KUKA KRL program: EPS_2_251349_MH88A_A_20250929014700.src

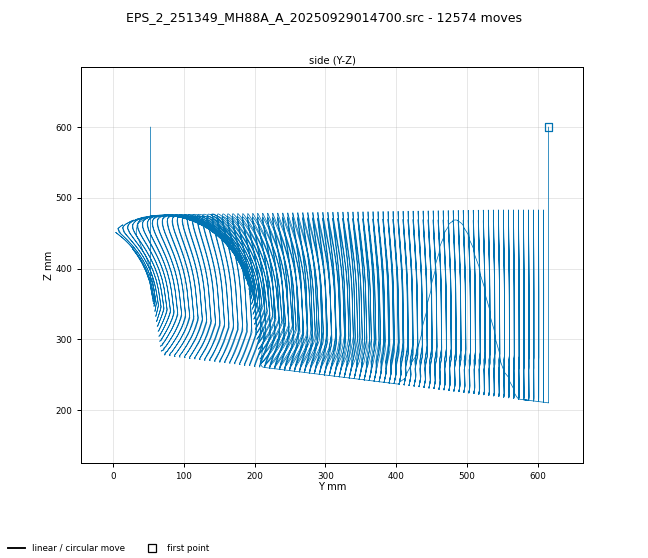
[picture p0: tool path of EPS_2_251349_MH88A_A_20250929014700.src, 12574 of 12576 moves have a stored position in this frame; points joined in program order, loops and branches not executed]
&ACCESS RVP
&REL 4
&COMMENT QRS 19112012
&PARAM EDITMASK = *
DEF PART()
EXT BAS (BAS_COMMAND :IN,REAL :IN )
INT I
BAS (#INITMOV,0 )

;KUKA QRS Post kuka4.cps  Date:22-06-2017 !

File_ID=2863

QRS_PRE_INIT()

;Init var - Until changes are made in qrs_pre_init
Outlet_Square_prg=0
Inlet_1_Square_prg=0
Inlet_2_Square_prg=0
Inlet_3_Square_prg=0
Inlet_4_Square_prg=0
Inlet_5_Square_prg=0

Outlet_1={X 0.000, Y 540.910, Z 382.500, B 0.000, E1 0.000 }
Inlet_1={X 0.000, Y 541.980, Z 367.500, B 0.000, E1 136.000 }
Outlet_1_type=201
Inlet_1_type=201
;QRS#1=Sidecore dimensions
;QRS#2=200-8" PVC SDR 35
;QRS#3=200-8" PVC SDR 35
;QRS#4=
;QRS#5=
;QRS#6=
;QRS#7=
;QRS#8=
;QRS#9=12-08 PSX
;QRS#10=12-08 PSX
;QRS#11=
;QRS#12=
;QRS#13=
;QRS#14=
;QRS#15=
;QRS#16=1220x127x762 2,5'
;QRS#17=EPS Height
;QRS#18=483
;QRS#19=*
;QRS#20= UPDATED VERSION 22-06-2017
;QRS#21=*
Outlet_Square=0100
Inlet_1_Square=0100
Inlet_2_Square=0
Inlet_3_Square=0
Inlet_4_Square=0
Inlet_5_Square=0
Mill_Square=1
Outlet_Square_Prg=204
Inlet_1_Square_prg=204

QRS_INIT()

$ADVANCE=5

; T1
PTP {E1 173.638,E2 173.638}
PTP {X 0,Y 615.435,A -85,B 0,C 180,E1 173.638,E2 173.638,E3 0,E4 0,E5 0,E6 0}
QRS_SPEED_INIT()
LIN {X 0,Y 615.435,Z 600,A -85,B 0,C 180,E1 173.638,E2 173.638,E3 0,E4 0,E5 0,E6 0} C_VEL
LIN {X 0,Y 615.435,Z 220.373,A -85,B 0,C 180,E1 173.638,E2 173.638} C_VEL
LIN {X 0,Y 615.435,Z 212.194,A -85,B 0,C 180,E1 173.638,E2 173.638} C_VEL
LIN {X 0,Y 615.43,Z 210.194,A -85,B 0,C 180,E1 173.452,E2 173.452} C_VEL
LIN {X 0,Y 615.434,Z 210.193,A -85,B 0,C 180,E1 171.468,E2 171.468} C_VEL
LIN {X 0,Y 615.439,Z 210.195,A -85,B 0,C 180,E1 169.126,E2 169.126} C_VEL
LIN {X 0,Y 615.455,Z 210.197,A -85,B 0,C 180,E1 166.803,E2 166.803} C_VEL
LIN {X 0,Y 615.495,Z 210.192,A -85,B 0,C 180,E1 164.101,E2 164.101} C_VEL
LIN {X 0,Y 615.456,Z 210.188,A -85,B 0,C 180,E1 161.359,E2 161.359} C_VEL
LIN {X 0,Y 615.456,Z 210.188,A -85,B 0,C 180,E1 159.274,E2 159.274} C_VEL
LIN {X 0,Y 615.456,Z 210.188,A -85,B 0,C 180,E1 157.161,E2 157.161} C_VEL
LIN {X 0,Y 615.455,Z 210.188,A -85,B 0,C 180,E1 155.013,E2 155.013} C_VEL
LIN {X 0,Y 615.492,Z 210.435,A -85,B 0,C 180,E1 154.019,E2 154.019} C_VEL
LIN {X 0,Y 615.489,Z 227.308,A -85,B 0,C 180,E1 151.349,E2 151.349} C_VEL
LIN {X 0,Y 615.432,Z 244.946,A -85,B 0,C 180,E1 148.617,E2 148.617} C_VEL
LIN {X 0,Y 615.462,Z 256.479,A -85,B 0,C 180,E1 146.868,E2 146.868} C_VEL
LIN {X 0,Y 615.457,Z 258.435,A -85,B 0,C 180,E1 146.794,E2 146.794} C_VEL
LIN {X 0,Y 615.498,Z 364.416,A -85,B 0,C 180,E1 145.533,E2 145.533} C_VEL
LIN {X 0,Y 615.498,Z 377.381,A -85,B 0,C 180,E1 145.244,E2 145.244} C_VEL
LIN {X 0,Y 615.498,Z 389.548,A -85,B 0,C 180,E1 144.844,E2 144.844} C_VEL
LIN {X 0,Y 615.482,Z 401.088,A -85,B 0,C 180,E1 144.335,E2 144.335} C_VEL
LIN {X 0,Y 615.475,Z 412.93,A -85,B 0,C 180,E1 143.656,E2 143.656} C_VEL
LIN {X 0,Y 615.498,Z 423.238,A -85,B 0,C 180,E1 142.913,E2 142.913} C_VEL
LIN {X 0,Y 615.495,Z 431.49,A -85,B 0,C 180,E1 142.181,E2 142.181} C_VEL
LIN {X 0,Y 615.496,Z 439.782,A -85,B 0,C 180,E1 141.315,E2 141.315} C_VEL
LIN {X 0,Y 615.497,Z 447.794,A -85,B 0,C 180,E1 140.26,E2 140.26} C_VEL
LIN {X 0,Y 615.496,Z 454.438,A -85,B 0,C 180,E1 139.154,E2 139.154} C_VEL
LIN {X 0,Y 615.495,Z 458.784,A -85,B 0,C 180,E1 138.227,E2 138.227} C_VEL
LIN {X 0,Y 615.494,Z 462.154,A -85,B 0,C 180,E1 137.304,E2 137.304} C_VEL
LIN {X 0,Y 615.493,Z 465.473,A -85,B 0,C 180,E1 136,E2 136} C_VEL
LIN {X 0,Y 615.493,Z 466.94,A -85,B 0,C 180,E1 134.942,E2 134.942} C_VEL
LIN {X 0,Y 615.492,Z 467.383,A -85,B 0,C 180,E1 134.008,E2 134.008} C_VEL
LIN {X 0,Y 615.489,Z 467.004,A -85,B 0,C 180,E1 133.058,E2 133.058} C_VEL
LIN {X 0,Y 615.494,Z 465.774,A -85,B 0,C 180,E1 132.092,E2 132.092} C_VEL
LIN {X 0,Y 615.495,Z 463.616,A -85,B 0,C 180,E1 131.106,E2 131.106} C_VEL
LIN {X 0,Y 615.497,Z 460.421,A -85,B 0,C 180,E1 130.101,E2 130.101} C_VEL
LIN {X 0,Y 615.493,Z 455.189,A -85,B 0,C 180,E1 128.902,E2 128.902} C_VEL
LIN {X 0,Y 615.494,Z 448.993,A -85,B 0,C 180,E1 127.828,E2 127.828} C_VEL
LIN {X 0,Y 615.495,Z 441.609,A -85,B 0,C 180,E1 126.818,E2 126.818} C_VEL
LIN {X 0,Y 615.497,Z 434.167,A -85,B 0,C 180,E1 125.991,E2 125.991} C_VEL
LIN {X 0,Y 615.498,Z 424.68,A -85,B 0,C 180,E1 125.112,E2 125.112} C_VEL
LIN {X 0,Y 615.494,Z 414.65,A -85,B 0,C 180,E1 124.367,E2 124.367} C_VEL
LIN {X 0,Y 615.48,Z 402.826,A -85,B 0,C 180,E1 123.666,E2 123.666} C_VEL
LIN {X 0,Y 615.497,Z 391.367,A -85,B 0,C 180,E1 123.136,E2 123.136} C_VEL
LIN {X 0,Y 615.498,Z 378.544,A -85,B 0,C 180,E1 122.698,E2 122.698} C_VEL
LIN {X 0,Y 615.497,Z 365.74,A -85,B 0,C 180,E1 122.401,E2 122.401} C_VEL
LIN {X 0,Y 615.477,Z 340.468,A -85,B 0,C 180,E1 122.078,E2 122.078} C_VEL
LIN {X 0,Y 615.431,Z 257.305,A -85,B 0,C 180,E1 121.092,E2 121.092} C_VEL
LIN {X 0,Y 615.435,Z 256.163,A -85,B 0,C 180,E1 121.006,E2 121.006} C_VEL
LIN {X 0,Y 615.491,Z 239.577,A -85,B 0,C 180,E1 118.467,E2 118.467} C_VEL
LIN {X 0,Y 615.479,Z 221.082,A -85,B 0,C 180,E1 115.585,E2 115.585} C_VEL
LIN {X 0,Y 615.488,Z 210.314,A -85,B 0,C 180,E1 113.851,E2 113.851} C_VEL
LIN {X 0,Y 615.454,Z 210.199,A -85,B 0,C 180,E1 111.432,E2 111.432} C_VEL
LIN {X 0,Y 615.451,Z 210.199,A -85,B 0,C 180,E1 109.338,E2 109.338} C_VEL
LIN {X 0,Y 615.448,Z 210.2,A -85,B 0,C 180,E1 107.27,E2 107.27} C_VEL
LIN {X 0,Y 615.408,Z 210.198,A -85,B 0,C 180,E1 104.55,E2 104.55} C_VEL
LIN {X 0,Y 615.407,Z 210.199,A -85,B 0,C 180,E1 102.53,E2 102.53} C_VEL
LIN {X 0,Y 615.408,Z 210.199,A -85,B 0,C 180,E1 100.527,E2 100.527} C_VEL
LIN {X 0,Y 615.41,Z 210.199,A -85,B 0,C 180,E1 98.536,E2 98.536} C_VEL
LIN {X 0,Y 615.414,Z 210.199,A -85,B 0,C 180,E1 96.556,E2 96.556} C_VEL
LIN {X 0,Y 615.421,Z 210.2,A -85,B 0,C 180,E1 94.584,E2 94.584} C_VEL
LIN {X 0,Y 615.43,Z 210.2,A -85,B 0,C 180,E1 92.617,E2 92.617} C_VEL
LIN {X 0,Y 615.441,Z 210.2,A -85,B 0,C 180,E1 90.653,E2 90.653} C_VEL
LIN {X 0,Y 615.402,Z 210.2,A -85,B 0,C 180,E1 88.036,E2 88.036} C_VEL
LIN {X 0,Y 615.406,Z 210.2,A -85,B 0,C 180,E1 86.07,E2 86.07} C_VEL
LIN {X 0,Y 615.412,Z 210.199,A -85,B 0,C 180,E1 84.1,E2 84.1} C_VEL
LIN {X 0,Y 615.42,Z 210.199,A -85,B 0,C 180,E1 82.123,E2 82.123} C_VEL
LIN {X 0,Y 615.429,Z 210.199,A -85,B 0,C 180,E1 80.136,E2 80.136} C_VEL
LIN {X 0,Y 615.438,Z 210.198,A -85,B 0,C 180,E1 78.137,E2 78.137} C_VEL
LIN {X 0,Y 615.438,Z 210.198,A -85,B 0,C 180,E1 76.052,E2 76.052} C_VEL
LIN {X 0,Y 615.407,Z 210.199,A -85,B 0,C 180,E1 73.41,E2 73.41} C_VEL
LIN {X 0,Y 615.408,Z 210.198,A -85,B 0,C 180,E1 71.351,E2 71.351} C_VEL
LIN {X 0,Y 615.407,Z 210.199,A -85,B 0,C 180,E1 69.266,E2 69.266} C_VEL
LIN {X 0,Y 615.408,Z 210.198,A -85,B 0,C 180,E1 67.151,E2 67.151} C_VEL
LIN {X 0,Y 615.412,Z 210.198,A -85,B 0,C 180,E1 65.004,E2 65.004} C_VEL
LIN {X 0,Y 615.48,Z 210.203,A -85,B 0,C 180,E1 62.084,E2 62.084} C_VEL
LIN {X 0,Y 615.499,Z 210.195,A -85,B 0,C 180,E1 59.84,E2 59.84} C_VEL
LIN {X 0,Y 615.468,Z 210.194,A -85,B 0,C 180,E1 57.541,E2 57.541} C_VEL
LIN {X 0,Y 615.436,Z 210.195,A -85,B 0,C 180,E1 55.181,E2 55.181} C_VEL
LIN {X 0,Y 615.418,Z 210.196,A -85,B 0,C 180,E1 52.752,E2 52.752} C_VEL
LIN {X 0,Y 615.457,Z 210.199,A -85,B 0,C 180,E1 49.903,E2 49.903} C_VEL
LIN {X 0,Y 615.446,Z 210.194,A -85,B 0,C 180,E1 46.946,E2 46.946} C_VEL
LIN {X 0,Y 615.424,Z 210.197,A -85,B 0,C 180,E1 44.145,E2 44.145} C_VEL
LIN {X 0,Y 615.425,Z 210.196,A -85,B 0,C 180,E1 42.073,E2 42.073} C_VEL
LIN {X 0,Y 615.44,Z 210.198,A -85,B 0,C 180,E1 39.745,E2 39.745} C_VEL
LIN {X 0,Y 615.487,Z 210.193,A -85,B 0,C 180,E1 36.936,E2 36.936} C_VEL
LIN {X 0,Y 615.477,Z 210.191,A -85,B 0,C 180,E1 34.698,E2 34.698} C_VEL
LIN {X 0,Y 615.444,Z 210.192,A -85,B 0,C 180,E1 32.324,E2 32.324} C_VEL
LIN {X 0,Y 615.438,Z 210.192,A -85,B 0,C 180,E1 30.155,E2 30.155} C_VEL
LIN {X 0,Y 615.431,Z 210.193,A -85,B 0,C 180,E1 27.911,E2 27.911} C_VEL
LIN {X 0,Y 615.429,Z 210.195,A -85,B 0,C 180,E1 25.557,E2 25.557} C_VEL
LIN {X 0,Y 615.481,Z 210.199,A -85,B 0,C 180,E1 22.838,E2 22.838} C_VEL
LIN {X 0,Y 615.465,Z 210.189,A -85,B 0,C 180,E1 20.028,E2 20.028} C_VEL
LIN {X 0,Y 615.461,Z 210.19,A -85,B 0,C 180,E1 17.952,E2 17.952} C_VEL
LIN {X 0,Y 615.469,Z 210.189,A -85,B 0,C 180,E1 15.9,E2 15.9} C_VEL
LIN {X 0,Y 615.475,Z 210.188,A -85,B 0,C 180,E1 13.869,E2 13.869} C_VEL
LIN {X 0,Y 615.433,Z 210.193,A -85,B 0,C 180,E1 11.189,E2 11.189} C_VEL
LIN {X 0,Y 615.437,Z 210.192,A -85,B 0,C 180,E1 9.195,E2 9.195} C_VEL
LIN {X 0,Y 615.441,Z 210.191,A -85,B 0,C 180,E1 7.211,E2 7.211} C_VEL
LIN {X 0,Y 615.447,Z 210.19,A -85,B 0,C 180,E1 5.237,E2 5.237} C_VEL
LIN {X 0,Y 615.456,Z 210.188,A -85,B 0,C 180,E1 3.269,E2 3.269} C_VEL
LIN {X 0,Y 615.468,Z 210.187,A -85,B 0,C 180,E1 1.304,E2 1.304} C_VEL
LIN {X 0,Y 615.439,Z 210.192,A -85,B 0,C 180,E1 -1.313,E2 -1.313} C_VEL
LIN {X 0,Y 615.466,Z 210.197,A -85,B 0,C 180,E1 -3.933,E2 -3.933} C_VEL
LIN {X 0,Y 615.493,Z 210.19,A -85,B 0,C 180,E1 -6.58,E2 -6.58} C_VEL
LIN {X 0,Y 615.46,Z 210.187,A -85,B 0,C 180,E1 -9.203,E2 -9.203} C_VEL
LIN {X 0,Y 615.468,Z 210.186,A -85,B 0,C 180,E1 -11.197,E2 -11.197} C_VEL
LIN {X 0,Y 615.474,Z 210.186,A -85,B 0,C 180,E1 -13.205,E2 -13.205} C_VEL
LIN {X 0,Y 615.482,Z 210.184,A -85,B 0,C 180,E1 -15.23,E2 -15.23} C_VEL
LIN {X 0,Y 615.446,Z 210.192,A -85,B 0,C 180,E1 -17.961,E2 -17.961} C_VEL
LIN {X 0,Y 615.489,Z 210.201,A -85,B 0,C 180,E1 -20.734,E2 -20.734} C_VEL
LIN {X 0,Y 615.48,Z 210.184,A -85,B 0,C 180,E1 -23.56,E2 -23.56} C_VEL
LIN {X 0,Y 615.474,Z 210.184,A -85,B 0,C 180,E1 -25.719,E2 -25.719} C_VEL
LIN {X 0,Y 615.464,Z 210.186,A -85,B 0,C 180,E1 -27.919,E2 -27.919} C_VEL
LIN {X 0,Y 615.455,Z 210.188,A -85,B 0,C 180,E1 -30.165,E2 -30.165} C_VEL
LIN {X 0,Y 615.451,Z 210.191,A -85,B 0,C 180,E1 -32.462,E2 -32.462} C_VEL
LIN {X 0,Y 615.459,Z 210.194,A -85,B 0,C 180,E1 -34.819,E2 -34.819} C_VEL
LIN {X 0,Y 615.484,Z 210.2,A -85,B 0,C 180,E1 -37.245,E2 -37.245} C_VEL
LIN {X 0,Y 615.496,Z 210.181,A -85,B 0,C 180,E1 -40.089,E2 -40.089} C_VEL
LIN {X 0,Y 615.473,Z 210.184,A -85,B 0,C 180,E1 -42.356,E2 -42.356} C_VEL
LIN {X 0,Y 615.455,Z 210.193,A -85,B 0,C 180,E1 -45.074,E2 -45.074} C_VEL
LIN {X 0,Y 615.487,Z 210.194,A -85,B 0,C 180,E1 -47.922,E2 -47.922} C_VEL
LIN {X 0,Y 615.49,Z 210.186,A -85,B 0,C 180,E1 -50.249,E2 -50.249} C_VEL
LIN {X 0,Y 615.478,Z 210.183,A -85,B 0,C 180,E1 -52.756,E2 -52.756} C_VEL
LIN {X 0,Y 615.458,Z 210.19,A -85,B 0,C 180,E1 -55.305,E2 -55.305} C_VEL
LIN {X 0,Y 615.466,Z 210.195,A -85,B 0,C 180,E1 -57.674,E2 -57.674} C_VEL
LIN {X 0,Y 615.494,Z 210.197,A -85,B 0,C 180,E1 -60.206,E2 -60.206} C_VEL
LIN {X 0,Y 615.497,Z 210.179,A -85,B 0,C 180,E1 -62.955,E2 -62.955} C_VEL
LIN {X 0,Y 615.462,Z 210.19,A -85,B 0,C 180,E1 -65.726,E2 -65.726} C_VEL
LIN {X 0,Y 615.489,Z 210.311,A -85,B 0,C 180,E1 -68.435,E2 -68.435} C_VEL
LIN {X 0,Y 615.496,Z 213.29,A -85,B 0,C 180,E1 -68.919,E2 -68.919} C_VEL
LIN {X 0,Y 615.486,Z 233.846,A -85,B 0,C 180,E1 -71.881,E2 -71.881} C_VEL
LIN {X 0,Y 615.474,Z 253.027,A -85,B 0,C 180,E1 -74.603,E2 -74.603} C_VEL
LIN {X 0,Y 615.487,Z 270.928,A -85,B 0,C 180,E1 -77.092,E2 -77.092} C_VEL
LIN {X 0,Y 615.488,Z 272.814,A -85,B 0,C 180,E1 -77.155,E2 -77.155} C_VEL
LIN {X 0,Y 615.498,Z 378.773,A -85,B 0,C 180,E1 -78.41,E2 -78.41} C_VEL
LIN {X 0,Y 615.498,Z 391.306,A -85,B 0,C 180,E1 -78.681,E2 -78.681} C_VEL
LIN {X 0,Y 615.496,Z 404.523,A -85,B 0,C 180,E1 -79.11,E2 -79.11} C_VEL
LIN {X 0,Y 615.491,Z 416.457,A -85,B 0,C 180,E1 -79.638,E2 -79.638} C_VEL
LIN {X 0,Y 615.48,Z 427.981,A -85,B 0,C 180,E1 -80.303,E2 -80.303} C_VEL
LIN {X 0,Y 615.499,Z 438.328,A -85,B 0,C 180,E1 -81.049,E2 -81.049} C_VEL
LIN {X 0,Y 615.497,Z 446.681,A -85,B 0,C 180,E1 -81.793,E2 -81.793} C_VEL
LIN {X 0,Y 615.498,Z 454.597,A -85,B 0,C 180,E1 -82.619,E2 -82.619} C_VEL
LIN {X 0,Y 615.49,Z 462.197,A -85,B 0,C 180,E1 -83.607,E2 -83.607} C_VEL
LIN {X 0,Y 615.498,Z 469.199,A -85,B 0,C 180,E1 -84.758,E2 -84.758} C_VEL
LIN {X 0,Y 615.493,Z 473.847,A -85,B 0,C 180,E1 -85.743,E2 -85.743} C_VEL
LIN {X 0,Y 615.494,Z 477.395,A -85,B 0,C 180,E1 -86.726,E2 -86.726} C_VEL
LIN {X 0,Y 615.497,Z 479.23,A -85,B 0,C 180,E1 -87.381,E2 -87.381} C_VEL
LIN {X 0,Y 615.497,Z 480.606,A -85,B 0,C 180,E1 -88.036,E2 -88.036} C_VEL
LIN {X 0,Y 615.496,Z 482.173,A -85,B 0,C 180,E1 -89.345,E2 -89.345} C_VEL
LIN {X 0,Y 615.494,Z 482.389,A -85,B 0,C 180,E1 -89.999,E2 -89.999} C_VEL
LIN {X 0,Y 615.495,Z 481.581,A -85,B 0,C 180,E1 -91.307,E2 -91.307} C_VEL
LIN {X 0,Y 615.497,Z 480.61,A -85,B 0,C 180,E1 -91.962,E2 -91.962} C_VEL
LIN {X 0,Y 615.497,Z 479.236,A -85,B 0,C 180,E1 -92.617,E2 -92.617} C_VEL
LIN {X 0,Y 615.496,Z 476.353,A -85,B 0,C 180,E1 -93.599,E2 -93.599} C_VEL
LIN {X 0,Y 615.498,Z 472.446,A -85,B 0,C 180,E1 -94.583,E2 -94.583} C_VEL
LIN {X 0,Y 615.499,Z 467.411,A -85,B 0,C 180,E1 -95.568,E2 -95.568} C_VEL
LIN {X 0,Y 615.489,Z 460.921,A -85,B 0,C 180,E1 -96.577,E2 -96.577} C_VEL
LIN {X 0,Y 615.497,Z 453.144,A -85,B 0,C 180,E1 -97.544,E2 -97.544} C_VEL
LIN {X 0,Y 615.498,Z 443.272,A -85,B 0,C 180,E1 -98.535,E2 -98.535} C_VEL
LIN {X 0,Y 615.495,Z 432.883,A -85,B 0,C 180,E1 -99.363,E2 -99.363} C_VEL
LIN {X 0,Y 615.475,Z 422.599,A -85,B 0,C 180,E1 -100.027,E2 -100.027} C_VEL
LIN {X 0,Y 615.497,Z 411.121,A -85,B 0,C 180,E1 -100.617,E2 -100.617} C_VEL
LIN {X 0,Y 615.499,Z 399.3,A -85,B 0,C 180,E1 -101.079,E2 -101.079} C_VEL
LIN {X 0,Y 615.498,Z 386.295,A -85,B 0,C 180,E1 -101.442,E2 -101.442} C_VEL
LIN {X 0,Y 615.5,Z 373.041,A -85,B 0,C 180,E1 -101.671,E2 -101.671} C_VEL
LIN {X 0,Y 615.488,Z 271.781,A -85,B 0,C 180,E1 -102.864,E2 -102.864} C_VEL
LIN {X 0,Y 615.485,Z 270.529,A -85,B 0,C 180,E1 -102.948,E2 -102.948} C_VEL
LIN {X 0,Y 615.481,Z 250.637,A -85,B 0,C 180,E1 -105.734,E2 -105.734} C_VEL
LIN {X 0,Y 615.491,Z 231.59,A -85,B 0,C 180,E1 -108.442,E2 -108.442} C_VEL
LIN {X 0,Y 615.492,Z 212.102,A -85,B 0,C 180,E1 -111.255,E2 -111.255} C_VEL
LIN {X 0,Y 615.49,Z 210.317,A -85,B 0,C 180,E1 -111.562,E2 -111.562} C_VEL
LIN {X 0,Y 615.461,Z 210.191,A -85,B 0,C 180,E1 -114.272,E2 -114.272} C_VEL
LIN {X 0,Y 615.457,Z 210.189,A -85,B 0,C 180,E1 -116.444,E2 -116.444} C_VEL
LIN {X 0,Y 615.459,Z 210.188,A -85,B 0,C 180,E1 -118.658,E2 -118.658} C_VEL
LIN {X 0,Y 615.485,Z 210.183,A -85,B 0,C 180,E1 -121.084,E2 -121.084} C_VEL
LIN {X 0,Y 615.483,Z 210.2,A -85,B 0,C 180,E1 -124.02,E2 -124.02} C_VEL
LIN {X 0,Y 615.456,Z 210.195,A -85,B 0,C 180,E1 -126.425,E2 -126.425} C_VEL
LIN {X 0,Y 615.453,Z 210.188,A -85,B 0,C 180,E1 -129.056,E2 -129.056} C_VEL
LIN {X 0,Y 615.479,Z 210.186,A -85,B 0,C 180,E1 -131.472,E2 -131.472} C_VEL
LIN {X 0,Y 615.495,Z 210.201,A -85,B 0,C 180,E1 -134.147,E2 -134.147} C_VEL
LIN {X 0,Y 615.443,Z 210.196,A -85,B 0,C 180,E1 -136.749,E2 -136.749} C_VEL
LIN {X 0,Y 615.438,Z 210.195,A -85,B 0,C 180,E1 -138.908,E2 -138.908} C_VEL
LIN {X 0,Y 615.432,Z 210.195,A -85,B 0,C 180,E1 -141.089,E2 -141.089} C_VEL
LIN {X 0,Y 615.439,Z 210.193,A -85,B 0,C 180,E1 -143.57,E2 -143.57} C_VEL
LIN {X 0,Y 615.467,Z 210.192,A -85,B 0,C 180,E1 -145.974,E2 -145.974} C_VEL
LIN {X 0,Y 615.445,Z 210.198,A -85,B 0,C 180,E1 -148.917,E2 -148.917} C_VEL
LIN {X 0,Y 615.418,Z 210.198,A -85,B 0,C 180,E1 -151.336,E2 -151.336} C_VEL
LIN {X 0,Y 615.414,Z 210.197,A -85,B 0,C 180,E1 -153.55,E2 -153.55} C_VEL
LIN {X 0,Y 615.425,Z 210.197,A -85,B 0,C 180,E1 -156,E2 -156} C_VEL
LIN {X 0,Y 615.48,Z 210.197,A -85,B 0,C 180,E1 -158.565,E2 -158.565} C_VEL
LIN {X 0,Y 615.419,Z 210.2,A -85,B 0,C 180,E1 -161.408,E2 -161.408} C_VEL
LIN {X 0,Y 615.41,Z 210.2,A -85,B 0,C 180,E1 -163.587,E2 -163.587} C_VEL
LIN {X 0,Y 615.424,Z 210.2,A -85,B 0,C 180,E1 -165.446,E2 -165.446} C_VEL
LIN {X 0,Y 615.433,Z 210.199,A -85,B 0,C 180,E1 -167.465,E2 -167.465} C_VEL
LIN {X 0,Y 615.442,Z 210.198,A -85,B 0,C 180,E1 -169.469,E2 -169.469} C_VEL
LIN {X 0,Y 615.412,Z 210.198,A -85,B 0,C 180,E1 -172.12,E2 -172.12} C_VEL
LIN {X 0,Y 615.416,Z 210.197,A -85,B 0,C 180,E1 -174.097,E2 -174.097} C_VEL
LIN {X 0,Y 615.421,Z 210.196,A -85,B 0,C 180,E1 -176.067,E2 -176.067} C_VEL
LIN {X 0,Y 615.429,Z 210.195,A -85,B 0,C 180,E1 -178.033,E2 -178.033} C_VEL
LIN {X 0,Y 615.438,Z 210.194,A -85,B 0,C 180,E1 -179.996,E2 -179.996} C_VEL
LIN {X 0,Y 615.449,Z 210.192,A -85,B 0,C 180,E1 -181.959,E2 -181.959} C_VEL
LIN {X 0,Y 615.462,Z 210.191,A -85,B 0,C 180,E1 -183.924,E2 -183.924} C_VEL
LIN {X 0,Y 615.43,Z 210.194,A -85,B 0,C 180,E1 -186.548,E2 -186.548} C_VEL
LIN {X 0,Y 614.774,Z 210.348,A -85,B 0,C 180,E1 -187.094,E2 -187.094} C_VEL
LIN {X 0,Y 611.95,Z 210.753,A -85,B 0,C 180,E1 -187.98,E2 -187.98} C_VEL
LIN {X 0,Y 609.559,Z 211.067,A -85,B 0,C 180,E1 -188.693,E2 -188.693} C_VEL
LIN {X 0,Y 608.529,Z 211.186,A -85,B 0,C 180,E1 -189.243,E2 -189.243} C_VEL
LIN {X 0,Y 608.444,Z 211.194,A -85,B 0,C 180,E1 -189.429,E2 -189.429} C_VEL
LIN {X 0,Y 608.456,Z 211.19,A -85,B 0,C 180,E1 -191.995,E2 -191.995} C_VEL
LIN {X 0,Y 608.44,Z 211.188,A -85,B 0,C 180,E1 -194.716,E2 -194.716} C_VEL
LIN {X 0,Y 608.442,Z 211.188,A -85,B 0,C 180,E1 -196.779,E2 -196.779} C_VEL
LIN {X 0,Y 608.434,Z 211.197,A -85,B 0,C 180,E1 -199.565,E2 -199.565} C_VEL
LIN {X 0,Y 608.46,Z 211.187,A -85,B 0,C 180,E1 -202.481,E2 -202.481} C_VEL
LIN {X 0,Y 608.438,Z 211.19,A -85,B 0,C 180,E1 -204.565,E2 -204.565} C_VEL
LIN {X 0,Y 608.493,Z 211.364,A -85,B 0,C 180,E1 -205.884,E2 -205.884} C_VEL
LIN {X 0,Y 608.508,Z 227.357,A -85,B 0,C 180,E1 -208.441,E2 -208.441} C_VEL
LIN {X 0,Y 608.429,Z 245.716,A -85,B 0,C 180,E1 -211.311,E2 -211.311} C_VEL
LIN {X 0,Y 608.473,Z 256.851,A -85,B 0,C 180,E1 -213.006,E2 -213.006} C_VEL
LIN {X 0,Y 608.548,Z 258.93,A -85,B 0,C 180,E1 -213.063,E2 -213.063} C_VEL
LIN {X 0,Y 608.571,Z 364.391,A -85,B 0,C 180,E1 -214.33,E2 -214.33} C_VEL
LIN {X 0,Y 608.552,Z 378.116,A -85,B 0,C 180,E1 -214.642,E2 -214.642} C_VEL
LIN {X 0,Y 608.525,Z 390.367,A -85,B 0,C 180,E1 -215.056,E2 -215.056} C_VEL
LIN {X 0,Y 608.488,Z 401.771,A -85,B 0,C 180,E1 -215.571,E2 -215.571} C_VEL
LIN {X 0,Y 608.484,Z 412.397,A -85,B 0,C 180,E1 -216.184,E2 -216.184} C_VEL
LIN {X 0,Y 608.472,Z 422.516,A -85,B 0,C 180,E1 -216.905,E2 -216.905} C_VEL
LIN {X 0,Y 608.476,Z 430.315,A -85,B 0,C 180,E1 -217.578,E2 -217.578} C_VEL
LIN {X 0,Y 608.452,Z 438.224,A -85,B 0,C 180,E1 -218.383,E2 -218.383} C_VEL
LIN {X 0,Y 608.437,Z 446.625,A -85,B 0,C 180,E1 -219.433,E2 -219.433} C_VEL
LIN {X 0,Y 608.433,Z 453.423,A -85,B 0,C 180,E1 -220.513,E2 -220.513} C_VEL
LIN {X 0,Y 608.446,Z 459.075,A -85,B 0,C 180,E1 -221.67,E2 -221.67} C_VEL
LIN {X 0,Y 608.457,Z 461.663,A -85,B 0,C 180,E1 -222.336,E2 -222.336} C_VEL
LIN {X 0,Y 608.428,Z 464.571,A -85,B 0,C 180,E1 -223.307,E2 -223.307} C_VEL
LIN {X 0,Y 608.418,Z 466.54,A -85,B 0,C 180,E1 -224.263,E2 -224.263} C_VEL
LIN {X 0,Y 608.414,Z 467.657,A -85,B 0,C 180,E1 -225.203,E2 -225.203} C_VEL
LIN {X 0,Y 608.419,Z 467.987,A -85,B 0,C 180,E1 -226.128,E2 -226.128} C_VEL
LIN {X 0,Y 608.424,Z 467.549,A -85,B 0,C 180,E1 -227.04,E2 -227.04} C_VEL
LIN {X 0,Y 608.421,Z 466.357,A -85,B 0,C 180,E1 -227.938,E2 -227.938} C_VEL
LIN {X 0,Y 608.429,Z 464.462,A -85,B 0,C 180,E1 -228.823,E2 -228.823} C_VEL
LIN {X 0,Y 608.442,Z 461.86,A -85,B 0,C 180,E1 -229.698,E2 -229.698} C_VEL
LIN {X 0,Y 608.435,Z 457.896,A -85,B 0,C 180,E1 -230.695,E2 -230.695} C_VEL
LIN {X 0,Y 608.434,Z 452.449,A -85,B 0,C 180,E1 -231.752,E2 -231.752} C_VEL
LIN {X 0,Y 608.437,Z 445.317,A -85,B 0,C 180,E1 -232.833,E2 -232.833} C_VEL
LIN {X 0,Y 608.469,Z 438.226,A -85,B 0,C 180,E1 -233.706,E2 -233.706} C_VEL
LIN {X 0,Y 608.478,Z 428.002,A -85,B 0,C 180,E1 -234.727,E2 -234.727} C_VEL
LIN {X 0,Y 608.484,Z 417.879,A -85,B 0,C 180,E1 -235.534,E2 -235.534} C_VEL
LIN {X 0,Y 608.474,Z 406.727,A -85,B 0,C 180,E1 -236.251,E2 -236.251} C_VEL
LIN {X 0,Y 608.518,Z 395.236,A -85,B 0,C 180,E1 -236.83,E2 -236.83} C_VEL
LIN {X 0,Y 608.533,Z 382.108,A -85,B 0,C 180,E1 -237.328,E2 -237.328} C_VEL
LIN {X 0,Y 608.562,Z 369.579,A -85,B 0,C 180,E1 -237.661,E2 -237.661} C_VEL
LIN {X 0,Y 608.57,Z 356.478,A -85,B 0,C 180,E1 -237.872,E2 -237.872} C_VEL
LIN {X 0,Y 608.462,Z 257.306,A -85,B 0,C 180,E1 -239.058,E2 -239.058} C_VEL
LIN {X 0,Y 608.442,Z 256.088,A -85,B 0,C 180,E1 -239.175,E2 -239.175} C_VEL
LIN {X 0,Y 608.486,Z 237.153,A -85,B 0,C 180,E1 -242.112,E2 -242.112} C_VEL
LIN {X 0,Y 608.503,Z 219.537,A -85,B 0,C 180,E1 -244.886,E2 -244.886} C_VEL
LIN {X 0,Y 608.481,Z 211.305,A -85,B 0,C 180,E1 -246.225,E2 -246.225} C_VEL
LIN {X 0,Y 608.392,Z 211.195,A -85,B 0,C 180,E1 -249.018,E2 -249.018} C_VEL
LIN {X 0,Y 608.404,Z 211.195,A -85,B 0,C 180,E1 -251.828,E2 -251.828} C_VEL
LIN {X 0,Y 608.434,Z 211.198,A -85,B 0,C 180,E1 -254.595,E2 -254.595} C_VEL
LIN {X 0,Y 608.407,Z 211.193,A -85,B 0,C 180,E1 -257.323,E2 -257.323} C_VEL
LIN {X 0,Y 608.394,Z 211.195,A -85,B 0,C 180,E1 -259.35,E2 -259.35} C_VEL
LIN {X 0,Y 608.389,Z 211.196,A -85,B 0,C 180,E1 -261.364,E2 -261.364} C_VEL
LIN {X 0,Y 608.391,Z 211.196,A -85,B 0,C 180,E1 -263.368,E2 -263.368} C_VEL
LIN {X 0,Y 608.394,Z 211.196,A -85,B 0,C 180,E1 -265.363,E2 -265.363} C_VEL
LIN {X 0,Y 608.421,Z 211.194,A -85,B 0,C 180,E1 -267.353,E2 -267.353} C_VEL
LIN {X 0,Y 608.389,Z 211.194,A -85,B 0,C 180,E1 -270.001,E2 -270.001} C_VEL
LIN {X 0,Y 608.419,Z 211.194,A -85,B 0,C 180,E1 -272.649,E2 -272.649} C_VEL
LIN {X 0,Y 608.47,Z 211.194,A -85,B 0,C 180,E1 -275.303,E2 -275.303} C_VEL
LIN {X 0,Y 608.408,Z 211.193,A -85,B 0,C 180,E1 -277.969,E2 -277.969} C_VEL
LIN {X 0,Y 608.394,Z 211.195,A -85,B 0,C 180,E1 -279.979,E2 -279.979} C_VEL
LIN {X 0,Y 608.403,Z 211.194,A -85,B 0,C 180,E1 -282.002,E2 -282.002} C_VEL
LIN {X 0,Y 608.405,Z 211.193,A -85,B 0,C 180,E1 -284.723,E2 -284.723} C_VEL
LIN {X 0,Y 608.413,Z 211.201,A -85,B 0,C 180,E1 -287.479,E2 -287.479} C_VEL
LIN {X 0,Y 608.41,Z 211.194,A -85,B 0,C 180,E1 -290.277,E2 -290.277} C_VEL
LIN {X 0,Y 608.39,Z 211.195,A -85,B 0,C 180,E1 -292.481,E2 -292.481} C_VEL
LIN {X 0,Y 608.397,Z 211.194,A -85,B 0,C 180,E1 -294.574,E2 -294.574} C_VEL
LIN {X 0,Y 608.409,Z 211.193,A -85,B 0,C 180,E1 -297.212,E2 -297.212} C_VEL
LIN {X 0,Y 608.473,Z 211.195,A -85,B 0,C 180,E1 -299.988,E2 -299.988} C_VEL
LIN {X 0,Y 608.407,Z 211.193,A -85,B 0,C 180,E1 -302.883,E2 -302.883} C_VEL
LIN {X 0,Y 608.387,Z 211.194,A -85,B 0,C 180,E1 -305.282,E2 -305.282} C_VEL
LIN {X 0,Y 608.437,Z 211.199,A -85,B 0,C 180,E1 -308.249,E2 -308.249} C_VEL
LIN {X 0,Y 608.459,Z 211.197,A -85,B 0,C 180,E1 -310.341,E2 -310.341} C_VEL
LIN {X 0,Y 608.418,Z 211.194,A -85,B 0,C 180,E1 -312.964,E2 -312.964} C_VEL
LIN {X 0,Y 608.398,Z 211.193,A -85,B 0,C 180,E1 -315.743,E2 -315.743} C_VEL
LIN {X 0,Y 608.405,Z 211.193,A -85,B 0,C 180,E1 -317.943,E2 -317.943} C_VEL
LIN {X 0,Y 608.458,Z 211.197,A -85,B 0,C 180,E1 -320.705,E2 -320.705} C_VEL
LIN {X 0,Y 608.454,Z 211.192,A -85,B 0,C 180,E1 -323.093,E2 -323.093} C_VEL
LIN {X 0,Y 608.443,Z 211.189,A -85,B 0,C 180,E1 -325.537,E2 -325.537} C_VEL
LIN {X 0,Y 608.421,Z 211.19,A -85,B 0,C 180,E1 -327.911,E2 -327.911} C_VEL
LIN {X 0,Y 608.413,Z 211.191,A -85,B 0,C 180,E1 -330.225,E2 -330.225} C_VEL
LIN {X 0,Y 608.433,Z 211.194,A -85,B 0,C 180,E1 -332.802,E2 -332.802} C_VEL
LIN {X 0,Y 608.449,Z 211.188,A -85,B 0,C 180,E1 -335.855,E2 -335.855} C_VEL
LIN {X 0,Y 608.429,Z 211.189,A -85,B 0,C 180,E1 -338.313,E2 -338.313} C_VEL
LIN {X 0,Y 608.411,Z 211.191,A -85,B 0,C 180,E1 -340.434,E2 -340.434} C_VEL
LIN {X 0,Y 608.41,Z 211.191,A -85,B 0,C 180,E1 -342.528,E2 -342.528} C_VEL
LIN {X 0,Y 608.431,Z 211.189,A -85,B 0,C 180,E1 -344.599,E2 -344.599} C_VEL
LIN {X 0,Y 608.454,Z 211.192,A -85,B 0,C 180,E1 -347.328,E2 -347.328} C_VEL
LIN {X 0,Y 608.458,Z 211.191,A -85,B 0,C 180,E1 -350.028,E2 -350.028} C_VEL
LIN {X 0,Y 608.42,Z 211.19,A -85,B 0,C 180,E1 -352.705,E2 -352.705} C_VEL
LIN {X 0,Y 608.433,Z 211.189,A -85,B 0,C 180,E1 -354.703,E2 -354.703} C_VEL
LIN {X 0,Y 608.438,Z 211.19,A -85,B 0,C 180,E1 -357.356,E2 -357.356} C_VEL
LIN {X 0,Y 608.474,Z 211.194,A -85,B 0,C 180,E1 -360.004,E2 -360.004} C_VEL
LIN {X 0,Y 608.48,Z 211.186,A -85,B 0,C 180,E1 -362.652,E2 -362.652} C_VEL
LIN {X 0,Y 608.429,Z 211.189,A -85,B 0,C 180,E1 -365.306,E2 -365.306} C_VEL
LIN {X 0,Y 608.426,Z 211.189,A -85,B 0,C 180,E1 -367.304,E2 -367.304} C_VEL
LIN {X 0,Y 608.429,Z 211.193,A -85,B 0,C 180,E1 -369.981,E2 -369.981} C_VEL
LIN {X 0,Y 608.476,Z 211.191,A -85,B 0,C 180,E1 -372.68,E2 -372.68} C_VEL
LIN {X 0,Y 608.458,Z 211.186,A -85,B 0,C 180,E1 -375.41,E2 -375.41} C_VEL
LIN {X 0,Y 608.422,Z 211.193,A -85,B 0,C 180,E1 -378.176,E2 -378.176} C_VEL
LIN {X 0,Y 608.461,Z 211.193,A -85,B 0,C 180,E1 -380.984,E2 -380.984} C_VEL
LIN {X 0,Y 608.442,Z 211.187,A -85,B 0,C 180,E1 -383.849,E2 -383.849} C_VEL
LIN {X 0,Y 608.428,Z 211.189,A -85,B 0,C 180,E1 -386.039,E2 -386.039} C_VEL
LIN {X 0,Y 608.421,Z 211.191,A -85,B 0,C 180,E1 -388.271,E2 -388.271} C_VEL
LIN {X 0,Y 608.435,Z 211.191,A -85,B 0,C 180,E1 -390.549,E2 -390.549} C_VEL
LIN {X 0,Y 608.447,Z 211.193,A -85,B 0,C 180,E1 -392.883,E2 -392.883} C_VEL
LIN {X 0,Y 608.438,Z 211.2,A -85,B 0,C 180,E1 -395.28,E2 -395.28} C_VEL
LIN {X 0,Y 608.469,Z 211.189,A -85,B 0,C 180,E1 -397.749,E2 -397.749} C_VEL
LIN {X 0,Y 608.449,Z 211.187,A -85,B 0,C 180,E1 -400.328,E2 -400.328} C_VEL
LIN {X 0,Y 608.426,Z 211.192,A -85,B 0,C 180,E1 -402.964,E2 -402.964} C_VEL
LIN {X 0,Y 608.457,Z 211.195,A -85,B 0,C 180,E1 -405.738,E2 -405.738} C_VEL
LIN {X 0,Y 608.45,Z 211.187,A -85,B 0,C 180,E1 -408.661,E2 -408.661} C_VEL
LIN {X 0,Y 608.427,Z 211.194,A -85,B 0,C 180,E1 -411.408,E2 -411.408} C_VEL
LIN {X 0,Y 608.453,Z 211.197,A -85,B 0,C 180,E1 -413.956,E2 -413.956} C_VEL
LIN {X 0,Y 608.456,Z 211.191,A -85,B 0,C 180,E1 -416.328,E2 -416.328} C_VEL
LIN {X 0,Y 608.456,Z 211.187,A -85,B 0,C 180,E1 -418.733,E2 -418.733} C_VEL
LIN {X 0,Y 608.455,Z 211.187,A -85,B 0,C 180,E1 -421.385,E2 -421.385} C_VEL
LIN {X 0,Y 608.44,Z 211.194,A -85,B 0,C 180,E1 -423.963,E2 -423.963} C_VEL
LIN {X 0,Y 608.451,Z 211.19,A -85,B 0,C 180,E1 -426.875,E2 -426.875} C_VEL
LIN {X 0,Y 608.471,Z 211.348,A -85,B 0,C 180,E1 -428.352,E2 -428.352} C_VEL
LIN {X 0,Y 608.512,Z 222.951,A -85,B 0,C 180,E1 -430.079,E2 -430.079} C_VEL
LIN {X 0,Y 608.52,Z 242.257,A -85,B 0,C 180,E1 -432.871,E2 -432.871} C_VEL
LIN {X 0,Y 608.482,Z 262.769,A -85,B 0,C 180,E1 -435.791,E2 -435.791} C_VEL
LIN {X 0,Y 608.497,Z 271.281,A -85,B 0,C 180,E1 -436.962,E2 -436.962} C_VEL
LIN {X 0,Y 608.588,Z 276.426,A -85,B 0,C 180,E1 -437.049,E2 -437.049} C_VEL
LIN {X 0,Y 608.549,Z 378.893,A -85,B 0,C 180,E1 -438.276,E2 -438.276} C_VEL
LIN {X 0,Y 608.549,Z 392.181,A -85,B 0,C 180,E1 -438.571,E2 -438.571} C_VEL
LIN {X 0,Y 608.546,Z 405.34,A -85,B 0,C 180,E1 -439.009,E2 -439.009} C_VEL
LIN {X 0,Y 608.516,Z 416.616,A -85,B 0,C 180,E1 -439.518,E2 -439.518} C_VEL
LIN {X 0,Y 608.468,Z 428.182,A -85,B 0,C 180,E1 -440.19,E2 -440.19} C_VEL
LIN {X 0,Y 608.485,Z 438.581,A -85,B 0,C 180,E1 -440.945,E2 -440.945} C_VEL
LIN {X 0,Y 608.459,Z 446.992,A -85,B 0,C 180,E1 -441.698,E2 -441.698} C_VEL
LIN {X 0,Y 608.471,Z 454.951,A -85,B 0,C 180,E1 -442.533,E2 -442.533} C_VEL
LIN {X 0,Y 608.438,Z 462.3,A -85,B 0,C 180,E1 -443.486,E2 -443.486} C_VEL
LIN {X 0,Y 608.45,Z 467.86,A -85,B 0,C 180,E1 -444.365,E2 -444.365} C_VEL
LIN {X 0,Y 608.432,Z 472.945,A -85,B 0,C 180,E1 -445.361,E2 -445.361} C_VEL
LIN {X 0,Y 608.449,Z 476.893,A -85,B 0,C 180,E1 -446.357,E2 -446.357} C_VEL
LIN {X 0,Y 608.425,Z 479.806,A -85,B 0,C 180,E1 -447.351,E2 -447.351} C_VEL
LIN {X 0,Y 608.442,Z 481.199,A -85,B 0,C 180,E1 -448.013,E2 -448.013} C_VEL
LIN {X 0,Y 608.439,Z 482.783,A -85,B 0,C 180,E1 -449.337,E2 -449.337} C_VEL
LIN {X 0,Y 608.434,Z 483,A -85,B 0,C 180,E1 -449.999,E2 -449.999} C_VEL
LIN {X 0,Y 608.448,Z 482.185,A -85,B 0,C 180,E1 -451.323,E2 -451.323} C_VEL
LIN {X 0,Y 608.442,Z 481.203,A -85,B 0,C 180,E1 -451.985,E2 -451.985} C_VEL
LIN {X 0,Y 608.425,Z 479.812,A -85,B 0,C 180,E1 -452.647,E2 -452.647} C_VEL
LIN {X 0,Y 608.449,Z 476.9,A -85,B 0,C 180,E1 -453.641,E2 -453.641} C_VEL
LIN {X 0,Y 608.432,Z 472.955,A -85,B 0,C 180,E1 -454.637,E2 -454.637} C_VEL
LIN {X 0,Y 608.437,Z 466.884,A -85,B 0,C 180,E1 -455.8,E2 -455.8} C_VEL
LIN {X 0,Y 608.461,Z 460.244,A -85,B 0,C 180,E1 -456.798,E2 -456.798} C_VEL
LIN {X 0,Y 608.456,Z 452,A -85,B 0,C 180,E1 -457.799,E2 -457.799} C_VEL
LIN {X 0,Y 608.477,Z 441.613,A -85,B 0,C 180,E1 -458.802,E2 -458.802} C_VEL
LIN {X 0,Y 608.486,Z 430.766,A -85,B 0,C 180,E1 -459.64,E2 -459.64} C_VEL
LIN {X 0,Y 608.489,Z 419.797,A -85,B 0,C 180,E1 -460.312,E2 -460.312} C_VEL
LIN {X 0,Y 608.536,Z 407.809,A -85,B 0,C 180,E1 -460.888,E2 -460.888} C_VEL
LIN {X 0,Y 608.533,Z 395.919,A -85,B 0,C 180,E1 -461.321,E2 -461.321} C_VEL
LIN {X 0,Y 608.542,Z 383.582,A -85,B 0,C 180,E1 -461.638,E2 -461.638} C_VEL
LIN {X 0,Y 608.574,Z 367.844,A -85,B 0,C 180,E1 -461.869,E2 -461.869} C_VEL
LIN {X 0,Y 608.547,Z 271.791,A -85,B 0,C 180,E1 -463.013,E2 -463.013} C_VEL
LIN {X 0,Y 608.459,Z 270.661,A -85,B 0,C 180,E1 -463.1,E2 -463.1} C_VEL
LIN {X 0,Y 608.494,Z 250.72,A -85,B 0,C 180,E1 -465.919,E2 -465.919} C_VEL
LIN {X 0,Y 608.516,Z 231.17,A -85,B 0,C 180,E1 -468.727,E2 -468.727} C_VEL
LIN {X 0,Y 608.549,Z 212.109,A -85,B 0,C 180,E1 -471.509,E2 -471.509} C_VEL
LIN {X 0,Y 608.478,Z 211.266,A -85,B 0,C 180,E1 -471.69,E2 -471.69} C_VEL
LIN {X 0,Y 608.444,Z 211.188,A -85,B 0,C 180,E1 -474.57,E2 -474.57} C_VEL
LIN {X 0,Y 608.486,Z 211.185,A -85,B 0,C 180,E1 -477.207,E2 -477.207} C_VEL
LIN {X 0,Y 608.451,Z 211.195,A -85,B 0,C 180,E1 -479.967,E2 -479.967} C_VEL
LIN {X 0,Y 608.434,Z 211.19,A -85,B 0,C 180,E1 -482.516,E2 -482.516} C_VEL
LIN {X 0,Y 608.423,Z 211.19,A -85,B 0,C 180,E1 -484.9,E2 -484.9} C_VEL
LIN {X 0,Y 608.465,Z 211.192,A -85,B 0,C 180,E1 -487.744,E2 -487.744} C_VEL
LIN {X 0,Y 608.439,Z 211.195,A -85,B 0,C 180,E1 -490.326,E2 -490.326} C_VEL
LIN {X 0,Y 608.413,Z 211.192,A -85,B 0,C 180,E1 -492.961,E2 -492.961} C_VEL
LIN {X 0,Y 608.418,Z 211.191,A -85,B 0,C 180,E1 -495.198,E2 -495.198} C_VEL
LIN {X 0,Y 608.475,Z 211.189,A -85,B 0,C 180,E1 -497.938,E2 -497.938} C_VEL
LIN {X 0,Y 608.419,Z 211.195,A -85,B 0,C 180,E1 -500.706,E2 -500.706} C_VEL
LIN {X 0,Y 608.4,Z 211.194,A -85,B 0,C 180,E1 -503.079,E2 -503.079} C_VEL
LIN {X 0,Y 608.427,Z 211.19,A -85,B 0,C 180,E1 -505.525,E2 -505.525} C_VEL
LIN {X 0,Y 608.435,Z 211.191,A -85,B 0,C 180,E1 -507.901,E2 -507.901} C_VEL
LIN {X 0,Y 608.46,Z 211.191,A -85,B 0,C 180,E1 -510.217,E2 -510.217} C_VEL
LIN {X 0,Y 608.395,Z 211.195,A -85,B 0,C 180,E1 -513.22,E2 -513.22} C_VEL
LIN {X 0,Y 608.404,Z 211.193,A -85,B 0,C 180,E1 -515.424,E2 -515.424} C_VEL
LIN {X 0,Y 608.438,Z 211.192,A -85,B 0,C 180,E1 -518.304,E2 -518.304} C_VEL
LIN {X 0,Y 608.407,Z 211.195,A -85,B 0,C 180,E1 -521.296,E2 -521.296} C_VEL
LIN {X 0,Y 608.386,Z 211.195,A -85,B 0,C 180,E1 -523.901,E2 -523.901} C_VEL
LIN {X 0,Y 608.433,Z 211.195,A -85,B 0,C 180,E1 -526.639,E2 -526.639} C_VEL
LIN {X 0,Y 608.434,Z 211.194,A -85,B 0,C 180,E1 -529.346,E2 -529.346} C_VEL
LIN {X 0,Y 608.385,Z 211.195,A -85,B 0,C 180,E1 -532.028,E2 -532.028} C_VEL
LIN {X 0,Y 608.398,Z 211.193,A -85,B 0,C 180,E1 -534.029,E2 -534.029} C_VEL
LIN {X 0,Y 608.394,Z 211.194,A -85,B 0,C 180,E1 -536.022,E2 -536.022} C_VEL
LIN {X 0,Y 608.403,Z 211.193,A -85,B 0,C 180,E1 -538.01,E2 -538.01} C_VEL
LIN {X 0,Y 608.431,Z 211.19,A -85,B 0,C 180,E1 -539.996,E2 -539.996} C_VEL
LIN {X 0,Y 608.418,Z 211.192,A -85,B 0,C 180,E1 -541.981,E2 -541.981} C_VEL
LIN {X 0,Y 608.428,Z 211.191,A -85,B 0,C 180,E1 -543.97,E2 -543.97} C_VEL
LIN {X 0,Y 608.414,Z 211.192,A -85,B 0,C 180,E1 -546.596,E2 -546.596} C_VEL
LIN {X 0,Y 608.411,Z 211.192,A -85,B 0,C 180,E1 -548.632,E2 -548.632} C_VEL
LIN {X 0,Y 608.444,Z 211.194,A -85,B 0,C 180,E1 -549.429,E2 -549.429} C_VEL
LIN {X 0,Y 607.775,Z 211.274,A -85,B 0,C 180,E1 -549.982,E2 -549.982} C_VEL
LIN {X 0,Y 604.929,Z 211.627,A -85,B 0,C 180,E1 -550.879,E2 -550.879} C_VEL
LIN {X 0,Y 602.521,Z 211.936,A -85,B 0,C 180,E1 -551.6,E2 -551.6} C_VEL
LIN {X 0,Y 601.478,Z 212.058,A -85,B 0,C 180,E1 -552.156,E2 -552.156} C_VEL
LIN {X 0,Y 601.389,Z 212.067,A -85,B 0,C 180,E1 -552.345,E2 -552.345} C_VEL
LIN {X 0,Y 601.398,Z 212.066,A -85,B 0,C 180,E1 -554.892,E2 -554.892} C_VEL
LIN {X 0,Y 601.402,Z 212.066,A -85,B 0,C 180,E1 -556.981,E2 -556.981} C_VEL
LIN {X 0,Y 601.391,Z 212.077,A -85,B 0,C 180,E1 -559.804,E2 -559.804} C_VEL
LIN {X 0,Y 601.42,Z 212.063,A -85,B 0,C 180,E1 -562.676,E2 -562.676} C_VEL
LIN {X 0,Y 601.381,Z 212.07,A -85,B 0,C 180,E1 -564.873,E2 -564.873} C_VEL
LIN {X 0,Y 601.458,Z 212.24,A -85,B 0,C 180,E1 -565.78,E2 -565.78} C_VEL
LIN {X 0,Y 601.482,Z 223.309,A -85,B 0,C 180,E1 -567.581,E2 -567.581} C_VEL
LIN {X 0,Y 601.412,Z 238.271,A -85,B 0,C 180,E1 -569.961,E2 -569.961} C_VEL
LIN {X 0,Y 601.433,Z 256.579,A -85,B 0,C 180,E1 -572.826,E2 -572.826} C_VEL
LIN {X 0,Y 601.625,Z 258.311,A -85,B 0,C 180,E1 -572.903,E2 -572.903} C_VEL
LIN {X 0,Y 601.611,Z 364.783,A -85,B 0,C 180,E1 -574.2,E2 -574.2} C_VEL
LIN {X 0,Y 601.596,Z 377.988,A -85,B 0,C 180,E1 -574.505,E2 -574.505} C_VEL
LIN {X 0,Y 601.557,Z 390.029,A -85,B 0,C 180,E1 -574.914,E2 -574.914} C_VEL
LIN {X 0,Y 601.502,Z 402.483,A -85,B 0,C 180,E1 -575.487,E2 -575.487} C_VEL
LIN {X 0,Y 601.476,Z 412.957,A -85,B 0,C 180,E1 -576.105,E2 -576.105} C_VEL
LIN {X 0,Y 601.452,Z 423.601,A -85,B 0,C 180,E1 -576.884,E2 -576.884} C_VEL
LIN {X 0,Y 601.43,Z 431.769,A -85,B 0,C 180,E1 -577.622,E2 -577.622} C_VEL
LIN {X 0,Y 601.393,Z 439.765,A -85,B 0,C 180,E1 -578.469,E2 -578.469} C_VEL
LIN {X 0,Y 601.378,Z 447.814,A -85,B 0,C 180,E1 -579.531,E2 -579.531} C_VEL
LIN {X 0,Y 601.344,Z 454.073,A -85,B 0,C 180,E1 -580.568,E2 -580.568} C_VEL
LIN {X 0,Y 601.362,Z 459.677,A -85,B 0,C 180,E1 -581.761,E2 -581.761} C_VEL
LIN {X 0,Y 601.353,Z 462.867,A -85,B 0,C 180,E1 -582.666,E2 -582.666} C_VEL
LIN {X 0,Y 601.33,Z 465.295,A -85,B 0,C 180,E1 -583.585,E2 -583.585} C_VEL
LIN {X 0,Y 601.331,Z 466.974,A -85,B 0,C 180,E1 -584.529,E2 -584.529} C_VEL
LIN {X 0,Y 601.332,Z 467.852,A -85,B 0,C 180,E1 -585.476,E2 -585.476} C_VEL
LIN {X 0,Y 601.327,Z 467.918,A -85,B 0,C 180,E1 -586.427,E2 -586.427} C_VEL
LIN {X 0,Y 601.337,Z 467.154,A -85,B 0,C 180,E1 -587.406,E2 -587.406} C_VEL
LIN {X 0,Y 601.344,Z 465.509,A -85,B 0,C 180,E1 -588.404,E2 -588.404} C_VEL
LIN {X 0,Y 601.332,Z 462.866,A -85,B 0,C 180,E1 -589.425,E2 -589.425} C_VEL
LIN {X 0,Y 601.349,Z 459.111,A -85,B 0,C 180,E1 -590.463,E2 -590.463} C_VEL
LIN {X 0,Y 601.339,Z 454.04,A -85,B 0,C 180,E1 -591.528,E2 -591.528} C_VEL
LIN {X 0,Y 601.381,Z 447.458,A -85,B 0,C 180,E1 -592.612,E2 -592.612} C_VEL
LIN {X 0,Y 601.383,Z 439.962,A -85,B 0,C 180,E1 -593.598,E2 -593.598} C_VEL
LIN {X 0,Y 601.423,Z 432.265,A -85,B 0,C 180,E1 -594.419,E2 -594.419} C_VEL
LIN {X 0,Y 601.436,Z 424.008,A -85,B 0,C 180,E1 -595.173,E2 -595.173} C_VEL
LIN {X 0,Y 601.466,Z 412.763,A -85,B 0,C 180,E1 -595.998,E2 -595.998} C_VEL
LIN {X 0,Y 601.496,Z 402.684,A -85,B 0,C 180,E1 -596.593,E2 -596.593} C_VEL
LIN {X 0,Y 601.556,Z 390.27,A -85,B 0,C 180,E1 -597.166,E2 -597.166} C_VEL
LIN {X 0,Y 601.59,Z 377.654,A -85,B 0,C 180,E1 -597.595,E2 -597.595} C_VEL
LIN {X 0,Y 601.618,Z 363.903,A -85,B 0,C 180,E1 -597.906,E2 -597.906} C_VEL
LIN {X 0,Y 601.451,Z 257.415,A -85,B 0,C 180,E1 -599.208,E2 -599.208} C_VEL
LIN {X 0,Y 601.421,Z 256.656,A -85,B 0,C 180,E1 -599.255,E2 -599.255} C_VEL
LIN {X 0,Y 601.483,Z 238.205,A -85,B 0,C 180,E1 -602.138,E2 -602.138} C_VEL
LIN {X 0,Y 601.508,Z 221.748,A -85,B 0,C 180,E1 -604.758,E2 -604.758} C_VEL
LIN {X 0,Y 601.421,Z 212.222,A -85,B 0,C 180,E1 -606.317,E2 -606.317} C_VEL
LIN {X 0,Y 601.36,Z 212.071,A -85,B 0,C 180,E1 -609.197,E2 -609.197} C_VEL
LIN {X 0,Y 601.361,Z 212.071,A -85,B 0,C 180,E1 -611.608,E2 -611.608} C_VEL
LIN {X 0,Y 601.38,Z 212.078,A -85,B 0,C 180,E1 -614.409,E2 -614.409} C_VEL
LIN {X 0,Y 601.36,Z 212.072,A -85,B 0,C 180,E1 -617.172,E2 -617.172} C_VEL
LIN {X 0,Y 601.369,Z 212.069,A -85,B 0,C 180,E1 -619.905,E2 -619.905} C_VEL
LIN {X 0,Y 601.4,Z 212.074,A -85,B 0,C 180,E1 -622.616,E2 -622.616} C_VEL
LIN {X 0,Y 601.366,Z 212.072,A -85,B 0,C 180,E1 -625.309,E2 -625.309} C_VEL
LIN {X 0,Y 601.386,Z 212.071,A -85,B 0,C 180,E1 -627.322,E2 -627.322} C_VEL
LIN {X 0,Y 601.358,Z 212.07,A -85,B 0,C 180,E1 -630.001,E2 -630.001} C_VEL
LIN {X 0,Y 601.384,Z 212.071,A -85,B 0,C 180,E1 -632.68,E2 -632.68} C_VEL
LIN {X 0,Y 601.421,Z 212.07,A -85,B 0,C 180,E1 -635.365,E2 -635.365} C_VEL
LIN {X 0,Y 601.369,Z 212.069,A -85,B 0,C 180,E1 -638.063,E2 -638.063} C_VEL
LIN {X 0,Y 601.358,Z 212.072,A -85,B 0,C 180,E1 -640.778,E2 -640.778} C_VEL
LIN {X 0,Y 601.372,Z 212.079,A -85,B 0,C 180,E1 -643.518,E2 -643.518} C_VEL
LIN {X 0,Y 601.386,Z 212.067,A -85,B 0,C 180,E1 -646.289,E2 -646.289} C_VEL
LIN {X 0,Y 601.355,Z 212.073,A -85,B 0,C 180,E1 -649.102,E2 -649.102} C_VEL
LIN {X 0,Y 601.363,Z 212.077,A -85,B 0,C 180,E1 -651.962,E2 -651.962} C_VEL
LIN {X 0,Y 601.4,Z 212.068,A -85,B 0,C 180,E1 -654.304,E2 -654.304} C_VEL
LIN {X 0,Y 601.383,Z 212.067,A -85,B 0,C 180,E1 -657.115,E2 -657.115} C_VEL
LIN {X 0,Y 601.432,Z 212.07,A -85,B 0,C 180,E1 -660.165,E2 -660.165} C_VEL
LIN {X 0,Y 601.378,Z 212.068,A -85,B 0,C 180,E1 -663.317,E2 -663.317} C_VEL
LIN {X 0,Y 601.395,Z 212.077,A -85,B 0,C 180,E1 -666.273,E2 -666.273} C_VEL
LIN {X 0,Y 601.362,Z 212.07,A -85,B 0,C 180,E1 -669.131,E2 -669.131} C_VEL
LIN {X 0,Y 601.377,Z 212.069,A -85,B 0,C 180,E1 -671.77,E2 -671.77} C_VEL
LIN {X 0,Y 601.375,Z 212.079,A -85,B 0,C 180,E1 -674.541,E2 -674.541} C_VEL
LIN {X 0,Y 601.371,Z 212.069,A -85,B 0,C 180,E1 -677.336,E2 -677.336} C_VEL
LIN {X 0,Y 601.372,Z 212.069,A -85,B 0,C 180,E1 -680.011,E2 -680.011} C_VEL
LIN {X 0,Y 601.407,Z 212.072,A -85,B 0,C 180,E1 -682.622,E2 -682.622} C_VEL
LIN {X 0,Y 601.426,Z 212.069,A -85,B 0,C 180,E1 -685.077,E2 -685.077} C_VEL
LIN {X 0,Y 601.401,Z 212.067,A -85,B 0,C 180,E1 -687.49,E2 -687.49} C_VEL
LIN {X 0,Y 601.375,Z 212.068,A -85,B 0,C 180,E1 -689.861,E2 -689.861} C_VEL
LIN {X 0,Y 601.373,Z 212.068,A -85,B 0,C 180,E1 -692.137,E2 -692.137} C_VEL
LIN {X 0,Y 601.371,Z 212.069,A -85,B 0,C 180,E1 -694.386,E2 -694.386} C_VEL
LIN {X 0,Y 601.368,Z 212.07,A -85,B 0,C 180,E1 -696.594,E2 -696.594} C_VEL
LIN {X 0,Y 601.428,Z 212.07,A -85,B 0,C 180,E1 -699.204,E2 -699.204} C_VEL
LIN {X 0,Y 601.41,Z 212.072,A -85,B 0,C 180,E1 -701.614,E2 -701.614} C_VEL
LIN {X 0,Y 601.383,Z 212.067,A -85,B 0,C 180,E1 -704.414,E2 -704.414} C_VEL
LIN {X 0,Y 601.395,Z 212.069,A -85,B 0,C 180,E1 -707.177,E2 -707.177} C_VEL
LIN {X 0,Y 601.43,Z 212.069,A -85,B 0,C 180,E1 -709.91,E2 -709.91} C_VEL
LIN {X 0,Y 601.393,Z 212.066,A -85,B 0,C 180,E1 -712.619,E2 -712.619} C_VEL
LIN {X 0,Y 601.404,Z 212.065,A -85,B 0,C 180,E1 -714.641,E2 -714.641} C_VEL
LIN {X 0,Y 601.407,Z 212.065,A -85,B 0,C 180,E1 -717.325,E2 -717.325} C_VEL
LIN {X 0,Y 601.443,Z 212.07,A -85,B 0,C 180,E1 -720.004,E2 -720.004} C_VEL
LIN {X 0,Y 601.442,Z 212.062,A -85,B 0,C 180,E1 -722.683,E2 -722.683} C_VEL
LIN {X 0,Y 601.396,Z 212.065,A -85,B 0,C 180,E1 -725.368,E2 -725.368} C_VEL
LIN {X 0,Y 601.378,Z 212.068,A -85,B 0,C 180,E1 -727.39,E2 -727.39} C_VEL
LIN {X 0,Y 601.395,Z 212.071,A -85,B 0,C 180,E1 -730.099,E2 -730.099} C_VEL
LIN {X 0,Y 601.417,Z 212.068,A -85,B 0,C 180,E1 -732.832,E2 -732.832} C_VEL
LIN {X 0,Y 601.397,Z 212.065,A -85,B 0,C 180,E1 -735.595,E2 -735.595} C_VEL
LIN {X 0,Y 601.383,Z 212.067,A -85,B 0,C 180,E1 -737.692,E2 -737.692} C_VEL
LIN {X 0,Y 601.392,Z 212.066,A -85,B 0,C 180,E1 -739.813,E2 -739.813} C_VEL
LIN {X 0,Y 601.418,Z 212.07,A -85,B 0,C 180,E1 -742.605,E2 -742.605} C_VEL
LIN {X 0,Y 601.418,Z 212.064,A -85,B 0,C 180,E1 -745.621,E2 -745.621} C_VEL
LIN {X 0,Y 601.377,Z 212.068,A -85,B 0,C 180,E1 -747.872,E2 -747.872} C_VEL
LIN {X 0,Y 601.413,Z 212.063,A -85,B 0,C 180,E1 -750.168,E2 -750.168} C_VEL
LIN {X 0,Y 601.406,Z 212.068,A -85,B 0,C 180,E1 -752.712,E2 -752.712} C_VEL
LIN {X 0,Y 601.386,Z 212.075,A -85,B 0,C 180,E1 -755.11,E2 -755.11} C_VEL
LIN {X 0,Y 601.444,Z 212.069,A -85,B 0,C 180,E1 -757.421,E2 -757.421} C_VEL
LIN {X 0,Y 601.414,Z 212.063,A -85,B 0,C 180,E1 -760.572,E2 -760.572} C_VEL
LIN {X 0,Y 601.382,Z 212.067,A -85,B 0,C 180,E1 -762.675,E2 -762.675} C_VEL
LIN {X 0,Y 601.414,Z 212.072,A -85,B 0,C 180,E1 -765.48,E2 -765.48} C_VEL
LIN {X 0,Y 601.423,Z 212.063,A -85,B 0,C 180,E1 -768.409,E2 -768.409} C_VEL
LIN {X 0,Y 601.399,Z 212.065,A -85,B 0,C 180,E1 -770.872,E2 -770.872} C_VEL
LIN {X 0,Y 601.394,Z 212.069,A -85,B 0,C 180,E1 -773.416,E2 -773.416} C_VEL
LIN {X 0,Y 601.426,Z 212.071,A -85,B 0,C 180,E1 -776.067,E2 -776.067} C_VEL
LIN {X 0,Y 601.428,Z 212.064,A -85,B 0,C 180,E1 -778.546,E2 -778.546} C_VEL
LIN {X 0,Y 601.414,Z 212.064,A -85,B 0,C 180,E1 -781.371,E2 -781.371} C_VEL
LIN {X 0,Y 601.4,Z 212.067,A -85,B 0,C 180,E1 -783.635,E2 -783.635} C_VEL
LIN {X 0,Y 601.422,Z 212.067,A -85,B 0,C 180,E1 -785.857,E2 -785.857} C_VEL
LIN {X 0,Y 601.453,Z 212.238,A -85,B 0,C 180,E1 -788.222,E2 -788.222} C_VEL
LIN {X 0,Y 601.612,Z 218.342,A -85,B 0,C 180,E1 -789.158,E2 -789.158} C_VEL
LIN {X 0,Y 601.53,Z 237.431,A -85,B 0,C 180,E1 -791.963,E2 -791.963} C_VEL
LIN {X 0,Y 601.451,Z 255.53,A -85,B 0,C 180,E1 -794.582,E2 -794.582} C_VEL
LIN {X 0,Y 601.461,Z 271.279,A -85,B 0,C 180,E1 -796.807,E2 -796.807} C_VEL
LIN {X 0,Y 601.67,Z 274.637,A -85,B 0,C 180,E1 -796.876,E2 -796.876} C_VEL
LIN {X 0,Y 601.621,Z 378.893,A -85,B 0,C 180,E1 -798.139,E2 -798.139} C_VEL
LIN {X 0,Y 601.593,Z 392.182,A -85,B 0,C 180,E1 -798.437,E2 -798.437} C_VEL
LIN {X 0,Y 601.552,Z 403.918,A -85,B 0,C 180,E1 -798.826,E2 -798.826} C_VEL
LIN {X 0,Y 601.531,Z 414.903,A -85,B 0,C 180,E1 -799.31,E2 -799.31} C_VEL
LIN {X 0,Y 601.462,Z 425.564,A -85,B 0,C 180,E1 -799.904,E2 -799.904} C_VEL
LIN {X 0,Y 601.447,Z 436.463,A -85,B 0,C 180,E1 -800.668,E2 -800.668} C_VEL
LIN {X 0,Y 601.424,Z 445.308,A -85,B 0,C 180,E1 -801.43,E2 -801.43} C_VEL
LIN {X 0,Y 601.397,Z 453.468,A -85,B 0,C 180,E1 -802.276,E2 -802.276} C_VEL
LIN {X 0,Y 601.384,Z 461.463,A -85,B 0,C 180,E1 -803.288,E2 -803.288} C_VEL
LIN {X 0,Y 601.372,Z 467.86,A -85,B 0,C 180,E1 -804.298,E2 -804.298} C_VEL
LIN {X 0,Y 601.336,Z 472.945,A -85,B 0,C 180,E1 -805.306,E2 -805.306} C_VEL
LIN {X 0,Y 601.368,Z 476.892,A -85,B 0,C 180,E1 -806.314,E2 -806.314} C_VEL
LIN {X 0,Y 601.325,Z 479.806,A -85,B 0,C 180,E1 -807.319,E2 -807.319} C_VEL
LIN {X 0,Y 601.341,Z 481.2,A -85,B 0,C 180,E1 -807.99,E2 -807.99} C_VEL
LIN {X 0,Y 601.339,Z 482.783,A -85,B 0,C 180,E1 -809.329,E2 -809.329} C_VEL
LIN {X 0,Y 601.335,Z 483,A -85,B 0,C 180,E1 -809.999,E2 -809.999} C_VEL
LIN {X 0,Y 601.347,Z 482.186,A -85,B 0,C 180,E1 -811.338,E2 -811.338} C_VEL
LIN {X 0,Y 601.341,Z 481.204,A -85,B 0,C 180,E1 -812.008,E2 -812.008} C_VEL
LIN {X 0,Y 601.325,Z 479.812,A -85,B 0,C 180,E1 -812.678,E2 -812.678} C_VEL
LIN {X 0,Y 601.367,Z 476.9,A -85,B 0,C 180,E1 -813.684,E2 -813.684} C_VEL
LIN {X 0,Y 601.336,Z 472.955,A -85,B 0,C 180,E1 -814.691,E2 -814.691} C_VEL
LIN {X 0,Y 601.372,Z 466.885,A -85,B 0,C 180,E1 -815.868,E2 -815.868} C_VEL
LIN {X 0,Y 601.381,Z 460.245,A -85,B 0,C 180,E1 -816.878,E2 -816.878} C_VEL
LIN {X 0,Y 601.4,Z 452.001,A -85,B 0,C 180,E1 -817.891,E2 -817.891} C_VEL
LIN {X 0,Y 601.435,Z 441.614,A -85,B 0,C 180,E1 -818.906,E2 -818.906} C_VEL
LIN {X 0,Y 601.472,Z 430.766,A -85,B 0,C 180,E1 -819.753,E2 -819.753} C_VEL
LIN {X 0,Y 601.495,Z 419.8,A -85,B 0,C 180,E1 -820.433,E2 -820.433} C_VEL
LIN {X 0,Y 601.551,Z 407.678,A -85,B 0,C 180,E1 -821.022,E2 -821.022} C_VEL
LIN {X 0,Y 601.578,Z 395.917,A -85,B 0,C 180,E1 -821.454,E2 -821.454} C_VEL
LIN {X 0,Y 601.608,Z 383.58,A -85,B 0,C 180,E1 -821.774,E2 -821.774} C_VEL
LIN {X 0,Y 601.643,Z 367.844,A -85,B 0,C 180,E1 -822.008,E2 -822.008} C_VEL
LIN {X 0,Y 601.574,Z 272.297,A -85,B 0,C 180,E1 -823.156,E2 -823.156} C_VEL
LIN {X 0,Y 601.453,Z 271.02,A -85,B 0,C 180,E1 -823.213,E2 -823.213} C_VEL
LIN {X 0,Y 601.485,Z 251.926,A -85,B 0,C 180,E1 -825.936,E2 -825.936} C_VEL
LIN {X 0,Y 601.531,Z 233.429,A -85,B 0,C 180,E1 -828.622,E2 -828.622} C_VEL
LIN {X 0,Y 601.645,Z 214.522,A -85,B 0,C 180,E1 -831.409,E2 -831.409} C_VEL
LIN {X 0,Y 601.436,Z 212.145,A -85,B 0,C 180,E1 -831.821,E2 -831.821} C_VEL
LIN {X 0,Y 601.405,Z 212.067,A -85,B 0,C 180,E1 -834.284,E2 -834.284} C_VEL
LIN {X 0,Y 601.455,Z 212.06,A -85,B 0,C 180,E1 -837.109,E2 -837.109} C_VEL
LIN {X 0,Y 601.403,Z 212.07,A -85,B 0,C 180,E1 -840.164,E2 -840.164} C_VEL
LIN {X 0,Y 601.403,Z 212.065,A -85,B 0,C 180,E1 -842.711,E2 -842.711} C_VEL
LIN {X 0,Y 601.382,Z 212.068,A -85,B 0,C 180,E1 -845.108,E2 -845.108} C_VEL
LIN {X 0,Y 601.431,Z 212.063,A -85,B 0,C 180,E1 -847.417,E2 -847.417} C_VEL
LIN {X 0,Y 601.4,Z 212.076,A -85,B 0,C 180,E1 -849.994,E2 -849.994} C_VEL
LIN {X 0,Y 601.373,Z 212.071,A -85,B 0,C 180,E1 -852.671,E2 -852.671} C_VEL
LIN {X 0,Y 601.397,Z 212.066,A -85,B 0,C 180,E1 -855.477,E2 -855.477} C_VEL
LIN {X 0,Y 601.411,Z 212.073,A -85,B 0,C 180,E1 -858.406,E2 -858.406} C_VEL
LIN {X 0,Y 601.383,Z 212.07,A -85,B 0,C 180,E1 -860.869,E2 -860.869} C_VEL
LIN {X 0,Y 601.385,Z 212.068,A -85,B 0,C 180,E1 -863.739,E2 -863.739} C_VEL
LIN {X 0,Y 601.413,Z 212.071,A -85,B 0,C 180,E1 -866.683,E2 -866.683} C_VEL
LIN {X 0,Y 601.381,Z 212.07,A -85,B 0,C 180,E1 -869.053,E2 -869.053} C_VEL
LIN {X 0,Y 601.376,Z 212.069,A -85,B 0,C 180,E1 -871.367,E2 -871.367} C_VEL
LIN {X 0,Y 601.387,Z 212.069,A -85,B 0,C 180,E1 -874.133,E2 -874.133} C_VEL
LIN {X 0,Y 601.366,Z 212.079,A -85,B 0,C 180,E1 -876.584,E2 -876.584} C_VEL
LIN {X 0,Y 601.374,Z 212.069,A -85,B 0,C 180,E1 -879.473,E2 -879.473} C_VEL
LIN {X 0,Y 601.34,Z 212.073,A -85,B 0,C 180,E1 -881.602,E2 -881.602} C_VEL
LIN {X 0,Y 601.374,Z 212.071,A -85,B 0,C 180,E1 -884.404,E2 -884.404} C_VEL
LIN {X 0,Y 601.362,Z 212.077,A -85,B 0,C 180,E1 -887.167,E2 -887.167} C_VEL
LIN {X 0,Y 601.395,Z 212.073,A -85,B 0,C 180,E1 -889.22,E2 -889.22} C_VEL
LIN {X 0,Y 601.367,Z 212.069,A -85,B 0,C 180,E1 -891.934,E2 -891.934} C_VEL
LIN {X 0,Y 601.354,Z 212.071,A -85,B 0,C 180,E1 -893.958,E2 -893.958} C_VEL
LIN {X 0,Y 601.351,Z 212.072,A -85,B 0,C 180,E1 -895.975,E2 -895.975} C_VEL
LIN {X 0,Y 601.377,Z 212.069,A -85,B 0,C 180,E1 -897.987,E2 -897.987} C_VEL
LIN {X 0,Y 601.402,Z 212.066,A -85,B 0,C 180,E1 -899.996,E2 -899.996} C_VEL
LIN {X 0,Y 601.395,Z 212.067,A -85,B 0,C 180,E1 -902.675,E2 -902.675} C_VEL
LIN {X 0,Y 601.42,Z 212.074,A -85,B 0,C 180,E1 -905.359,E2 -905.359} C_VEL
LIN {X 0,Y 601.421,Z 212.064,A -85,B 0,C 180,E1 -908.056,E2 -908.056} C_VEL
LIN {X 0,Y 601.387,Z 212.069,A -85,B 0,C 180,E1 -911.003,E2 -911.003} C_VEL
LIN {X 0,Y 601.389,Z 212.067,A -85,B 0,C 180,E1 -912.345,E2 -912.345} C_VEL
LIN {X 0,Y 600.71,Z 212.153,A -85,B 0,C 180,E1 -912.904,E2 -912.904} C_VEL
LIN {X 0,Y 597.854,Z 212.514,A -85,B 0,C 180,E1 -913.812,E2 -913.812} C_VEL
LIN {X 0,Y 595.451,Z 212.811,A -85,B 0,C 180,E1 -914.543,E2 -914.543} C_VEL
LIN {X 0,Y 594.423,Z 212.937,A -85,B 0,C 180,E1 -915.107,E2 -915.107} C_VEL
LIN {X 0,Y 594.341,Z 212.948,A -85,B 0,C 180,E1 -915.297,E2 -915.297} C_VEL
LIN {X 0,Y 594.361,Z 212.95,A -85,B 0,C 180,E1 -917.899,E2 -917.899} C_VEL
LIN {X 0,Y 594.352,Z 212.944,A -85,B 0,C 180,E1 -920.915,E2 -920.915} C_VEL
LIN {X 0,Y 594.375,Z 212.95,A -85,B 0,C 180,E1 -923.698,E2 -923.698} C_VEL
LIN {X 0,Y 594.39,Z 213.139,A -85,B 0,C 180,E1 -925.678,E2 -925.678} C_VEL
LIN {X 0,Y 594.576,Z 219.155,A -85,B 0,C 180,E1 -926.683,E2 -926.683} C_VEL
LIN {X 0,Y 594.448,Z 235.828,A -85,B 0,C 180,E1 -929.376,E2 -929.376} C_VEL
LIN {X 0,Y 594.387,Z 253.164,A -85,B 0,C 180,E1 -932.138,E2 -932.138} C_VEL
LIN {X 0,Y 594.42,Z 256.786,A -85,B 0,C 180,E1 -932.688,E2 -932.688} C_VEL
LIN {X 0,Y 594.733,Z 259.533,A -85,B 0,C 180,E1 -932.764,E2 -932.764} C_VEL
LIN {X 0,Y 594.668,Z 364.29,A -85,B 0,C 180,E1 -934.051,E2 -934.051} C_VEL
LIN {X 0,Y 594.634,Z 378.164,A -85,B 0,C 180,E1 -934.372,E2 -934.372} C_VEL
LIN {X 0,Y 594.588,Z 390.86,A -85,B 0,C 180,E1 -934.815,E2 -934.815} C_VEL
LIN {X 0,Y 594.513,Z 403.002,A -85,B 0,C 180,E1 -935.39,E2 -935.39} C_VEL
LIN {X 0,Y 594.468,Z 413.418,A -85,B 0,C 180,E1 -936.018,E2 -936.018} C_VEL
LIN {X 0,Y 594.425,Z 423.34,A -85,B 0,C 180,E1 -936.754,E2 -936.754} C_VEL
LIN {X 0,Y 594.375,Z 431.203,A -85,B 0,C 180,E1 -937.463,E2 -937.463} C_VEL
LIN {X 0,Y 594.32,Z 439.666,A -85,B 0,C 180,E1 -938.368,E2 -938.368} C_VEL
LIN {X 0,Y 594.291,Z 446.357,A -85,B 0,C 180,E1 -939.239,E2 -939.239} C_VEL
LIN {X 0,Y 594.287,Z 453.269,A -85,B 0,C 180,E1 -940.352,E2 -940.352} C_VEL
LIN {X 0,Y 594.262,Z 458.652,A -85,B 0,C 180,E1 -941.465,E2 -941.465} C_VEL
LIN {X 0,Y 594.273,Z 462.085,A -85,B 0,C 180,E1 -942.374,E2 -942.374} C_VEL
LIN {X 0,Y 594.257,Z 464.717,A -85,B 0,C 180,E1 -943.3,E2 -943.3} C_VEL
LIN {X 0,Y 594.219,Z 466.578,A -85,B 0,C 180,E1 -944.241,E2 -944.241} C_VEL
LIN {X 0,Y 594.218,Z 467.671,A -85,B 0,C 180,E1 -945.195,E2 -945.195} C_VEL
LIN {X 0,Y 594.224,Z 467.979,A -85,B 0,C 180,E1 -946.164,E2 -946.164} C_VEL
LIN {X 0,Y 594.25,Z 467.462,A -85,B 0,C 180,E1 -947.149,E2 -947.149} C_VEL
LIN {X 0,Y 594.235,Z 465.313,A -85,B 0,C 180,E1 -948.526,E2 -948.526} C_VEL
LIN {X 0,Y 594.248,Z 462.992,A -85,B 0,C 180,E1 -949.425,E2 -949.425} C_VEL
LIN {X 0,Y 594.265,Z 459.949,A -85,B 0,C 180,E1 -950.313,E2 -950.313} C_VEL
LIN {X 0,Y 594.266,Z 455.589,A -85,B 0,C 180,E1 -951.298,E2 -951.298} C_VEL
LIN {X 0,Y 594.272,Z 449.405,A -85,B 0,C 180,E1 -952.394,E2 -952.394} C_VEL
LIN {X 0,Y 594.325,Z 441.398,A -85,B 0,C 180,E1 -953.512,E2 -953.512} C_VEL
LIN {X 0,Y 594.378,Z 433.584,A -85,B 0,C 180,E1 -954.387,E2 -954.387} C_VEL
LIN {X 0,Y 594.409,Z 424.779,A -85,B 0,C 180,E1 -955.218,E2 -955.218} C_VEL
LIN {X 0,Y 594.451,Z 414.132,A -85,B 0,C 180,E1 -956.024,E2 -956.024} C_VEL
LIN {X 0,Y 594.488,Z 403.845,A -85,B 0,C 180,E1 -956.655,E2 -956.655} C_VEL
LIN {X 0,Y 594.572,Z 391.106,A -85,B 0,C 180,E1 -957.265,E2 -957.265} C_VEL
LIN {X 0,Y 594.642,Z 378.027,A -85,B 0,C 180,E1 -957.721,E2 -957.721} C_VEL
LIN {X 0,Y 594.693,Z 364.593,A -85,B 0,C 180,E1 -958.034,E2 -958.034} C_VEL
LIN {X 0,Y 594.522,Z 257.953,A -85,B 0,C 180,E1 -959.352,E2 -959.352} C_VEL
LIN {X 0,Y 594.378,Z 256.437,A -85,B 0,C 180,E1 -959.442,E2 -959.442} C_VEL
LIN {X 0,Y 594.47,Z 239.344,A -85,B 0,C 180,E1 -962.15,E2 -962.15} C_VEL
LIN {X 0,Y 594.523,Z 222.801,A -85,B 0,C 180,E1 -964.815,E2 -964.815} C_VEL
LIN {X 0,Y 594.434,Z 213.228,A -85,B 0,C 180,E1 -966.392,E2 -966.392} C_VEL
LIN {X 0,Y 594.353,Z 212.948,A -85,B 0,C 180,E1 -967.034,E2 -967.034} C_VEL
LIN {X 0,Y 594.32,Z 212.952,A -85,B 0,C 180,E1 -969.946,E2 -969.946} C_VEL
LIN {X 0,Y 594.326,Z 212.951,A -85,B 0,C 180,E1 -972.806,E2 -972.806} C_VEL
LIN {X 0,Y 594.343,Z 212.945,A -85,B 0,C 180,E1 -975.81,E2 -975.81} C_VEL
LIN {X 0,Y 594.371,Z 212.947,A -85,B 0,C 180,E1 -978.892,E2 -978.892} C_VEL
LIN {X 0,Y 594.344,Z 212.944,A -85,B 0,C 180,E1 -981.844,E2 -981.844} C_VEL
LIN {X 0,Y 594.374,Z 212.947,A -85,B 0,C 180,E1 -984.573,E2 -984.573} C_VEL
LIN {X 0,Y 594.351,Z 212.948,A -85,B 0,C 180,E1 -987.29,E2 -987.29} C_VEL
LIN {X 0,Y 594.327,Z 212.946,A -85,B 0,C 180,E1 -990.001,E2 -990.001} C_VEL
LIN {X 0,Y 594.349,Z 212.948,A -85,B 0,C 180,E1 -992.712,E2 -992.712} C_VEL
LIN {X 0,Y 594.374,Z 212.947,A -85,B 0,C 180,E1 -995.429,E2 -995.429} C_VEL
LIN {X 0,Y 594.344,Z 212.944,A -85,B 0,C 180,E1 -998.159,E2 -998.159} C_VEL
LIN {X 0,Y 594.372,Z 212.947,A -85,B 0,C 180,E1 -1001.108,E2 -1001.108} C_VEL
LIN {X 0,Y 594.339,Z 212.945,A -85,B 0,C 180,E1 -1004.188,E2 -1004.188} C_VEL
LIN {X 0,Y 594.329,Z 212.95,A -85,B 0,C 180,E1 -1007.196,E2 -1007.196} C_VEL
LIN {X 0,Y 594.32,Z 212.952,A -85,B 0,C 180,E1 -1010.057,E2 -1010.057} C_VEL
LIN {X 0,Y 594.302,Z 212.949,A -85,B 0,C 180,E1 -1012.971,E2 -1012.971} C_VEL
LIN {X 0,Y 594.325,Z 212.947,A -85,B 0,C 180,E1 -1015.196,E2 -1015.196} C_VEL
LIN {X 0,Y 594.317,Z 212.951,A -85,B 0,C 180,E1 -1017.531,E2 -1017.531} C_VEL
LIN {X 0,Y 594.368,Z 212.947,A -85,B 0,C 180,E1 -1020.341,E2 -1020.341} C_VEL
LIN {X 0,Y 594.328,Z 212.946,A -85,B 0,C 180,E1 -1022.954,E2 -1022.954} C_VEL
LIN {X 0,Y 594.326,Z 212.946,A -85,B 0,C 180,E1 -1025.411,E2 -1025.411} C_VEL
LIN {X 0,Y 594.345,Z 212.949,A -85,B 0,C 180,E1 -1027.945,E2 -1027.945} C_VEL
LIN {X 0,Y 594.346,Z 212.947,A -85,B 0,C 180,E1 -1030.83,E2 -1030.83} C_VEL
LIN {X 0,Y 594.326,Z 212.946,A -85,B 0,C 180,E1 -1033.304,E2 -1033.304} C_VEL
LIN {X 0,Y 594.338,Z 212.949,A -85,B 0,C 180,E1 -1036.164,E2 -1036.164} C_VEL
LIN {X 0,Y 594.349,Z 212.946,A -85,B 0,C 180,E1 -1039.182,E2 -1039.182} C_VEL
LIN {X 0,Y 594.345,Z 212.945,A -85,B 0,C 180,E1 -1042.065,E2 -1042.065} C_VEL
LIN {X 0,Y 594.353,Z 212.951,A -85,B 0,C 180,E1 -1044.677,E2 -1044.677} C_VEL
LIN {X 0,Y 594.347,Z 212.952,A -85,B 0,C 180,E1 -1047.094,E2 -1047.094} C_VEL
LIN {X 0,Y 594.344,Z 212.945,A -85,B 0,C 180,E1 -1049.68,E2 -1049.68} C_VEL
LIN {X 0,Y 594.356,Z 212.943,A -85,B 0,C 180,E1 -1051.779,E2 -1051.779} C_VEL
LIN {X 0,Y 594.335,Z 212.945,A -85,B 0,C 180,E1 -1054.061,E2 -1054.061} C_VEL
LIN {X 0,Y 594.349,Z 212.943,A -85,B 0,C 180,E1 -1056.301,E2 -1056.301} C_VEL
LIN {X 0,Y 594.396,Z 212.946,A -85,B 0,C 180,E1 -1059.23,E2 -1059.23} C_VEL
LIN {X 0,Y 594.33,Z 212.947,A -85,B 0,C 180,E1 -1062.1,E2 -1062.1} C_VEL
LIN {X 0,Y 594.343,Z 212.945,A -85,B 0,C 180,E1 -1064.224,E2 -1064.224} C_VEL
LIN {X 0,Y 594.359,Z 212.943,A -85,B 0,C 180,E1 -1066.326,E2 -1066.326} C_VEL
LIN {X 0,Y 594.358,Z 212.943,A -85,B 0,C 180,E1 -1068.944,E2 -1068.944} C_VEL
LIN {X 0,Y 594.407,Z 212.947,A -85,B 0,C 180,E1 -1071.848,E2 -1071.848} C_VEL
LIN {X 0,Y 594.373,Z 212.941,A -85,B 0,C 180,E1 -1074.577,E2 -1074.577} C_VEL
LIN {X 0,Y 594.376,Z 212.941,A -85,B 0,C 180,E1 -1077.294,E2 -1077.294} C_VEL
LIN {X 0,Y 594.411,Z 212.946,A -85,B 0,C 180,E1 -1080.004,E2 -1080.004} C_VEL
LIN {X 0,Y 594.405,Z 212.938,A -85,B 0,C 180,E1 -1082.715,E2 -1082.715} C_VEL
LIN {X 0,Y 594.363,Z 212.942,A -85,B 0,C 180,E1 -1085.432,E2 -1085.432} C_VEL
LIN {X 0,Y 594.359,Z 212.95,A -85,B 0,C 180,E1 -1088.161,E2 -1088.161} C_VEL
LIN {X 0,Y 594.4,Z 212.938,A -85,B 0,C 180,E1 -1091.076,E2 -1091.076} C_VEL
LIN {X 0,Y 594.372,Z 212.945,A -85,B 0,C 180,E1 -1094.165,E2 -1094.165} C_VEL
LIN {X 0,Y 594.382,Z 212.941,A -85,B 0,C 180,E1 -1097.197,E2 -1097.197} C_VEL
LIN {X 0,Y 594.364,Z 212.942,A -85,B 0,C 180,E1 -1100.057,E2 -1100.057} C_VEL
LIN {X 0,Y 594.362,Z 212.951,A -85,B 0,C 180,E1 -1102.971,E2 -1102.971} C_VEL
LIN {X 0,Y 594.354,Z 212.942,A -85,B 0,C 180,E1 -1105.948,E2 -1105.948} C_VEL
LIN {X 0,Y 594.335,Z 212.945,A -85,B 0,C 180,E1 -1108.232,E2 -1108.232} C_VEL
LIN {X 0,Y 594.377,Z 212.942,A -85,B 0,C 180,E1 -1110.563,E2 -1110.563} C_VEL
LIN {X 0,Y 594.385,Z 212.946,A -85,B 0,C 180,E1 -1112.952,E2 -1112.952} C_VEL
LIN {X 0,Y 594.336,Z 212.954,A -85,B 0,C 180,E1 -1115.413,E2 -1115.413} C_VEL
LIN {X 0,Y 594.388,Z 212.94,A -85,B 0,C 180,E1 -1117.943,E2 -1117.943} C_VEL
LIN {X 0,Y 594.375,Z 212.942,A -85,B 0,C 180,E1 -1120.821,E2 -1120.821} C_VEL
LIN {X 0,Y 594.356,Z 212.949,A -85,B 0,C 180,E1 -1123.303,E2 -1123.303} C_VEL
LIN {X 0,Y 594.358,Z 212.945,A -85,B 0,C 180,E1 -1126.164,E2 -1126.164} C_VEL
LIN {X 0,Y 594.38,Z 212.94,A -85,B 0,C 180,E1 -1128.535,E2 -1128.535} C_VEL
LIN {X 0,Y 594.378,Z 212.942,A -85,B 0,C 180,E1 -1131.299,E2 -1131.299} C_VEL
LIN {X 0,Y 594.355,Z 212.951,A -85,B 0,C 180,E1 -1133.755,E2 -1133.755} C_VEL
LIN {X 0,Y 594.373,Z 212.947,A -85,B 0,C 180,E1 -1136.238,E2 -1136.238} C_VEL
LIN {X 0,Y 594.376,Z 212.942,A -85,B 0,C 180,E1 -1138.649,E2 -1138.649} C_VEL
LIN {X 0,Y 594.385,Z 212.939,A -85,B 0,C 180,E1 -1141.044,E2 -1141.044} C_VEL
LIN {X 0,Y 594.388,Z 212.939,A -85,B 0,C 180,E1 -1143.3,E2 -1143.3} C_VEL
LIN {X 0,Y 594.357,Z 212.944,A -85,B 0,C 180,E1 -1145.575,E2 -1145.575} C_VEL
LIN {X 0,Y 594.397,Z 213.132,A -85,B 0,C 180,E1 -1148.087,E2 -1148.087} C_VEL
LIN {X 0,Y 594.696,Z 216.838,A -85,B 0,C 180,E1 -1148.678,E2 -1148.678} C_VEL
LIN {X 0,Y 594.575,Z 236.224,A -85,B 0,C 180,E1 -1151.566,E2 -1151.566} C_VEL
LIN {X 0,Y 594.487,Z 254.323,A -85,B 0,C 180,E1 -1154.221,E2 -1154.221} C_VEL
LIN {X 0,Y 594.43,Z 271.277,A -85,B 0,C 180,E1 -1156.648,E2 -1156.648} C_VEL
LIN {X 0,Y 594.769,Z 274.637,A -85,B 0,C 180,E1 -1156.721,E2 -1156.721} C_VEL
LIN {X 0,Y 594.674,Z 378.893,A -85,B 0,C 180,E1 -1157.998,E2 -1157.998} C_VEL
LIN {X 0,Y 594.641,Z 392.183,A -85,B 0,C 180,E1 -1158.3,E2 -1158.3} C_VEL
LIN {X 0,Y 594.59,Z 405.368,A -85,B 0,C 180,E1 -1158.749,E2 -1158.749} C_VEL
LIN {X 0,Y 594.538,Z 416.613,A -85,B 0,C 180,E1 -1159.269,E2 -1159.269} C_VEL
LIN {X 0,Y 594.456,Z 428.185,A -85,B 0,C 180,E1 -1159.956,E2 -1159.956} C_VEL
LIN {X 0,Y 594.414,Z 438.584,A -85,B 0,C 180,E1 -1160.729,E2 -1160.729} C_VEL
LIN {X 0,Y 594.349,Z 447.021,A -85,B 0,C 180,E1 -1161.499,E2 -1161.499} C_VEL
LIN {X 0,Y 594.348,Z 454.951,A -85,B 0,C 180,E1 -1162.354,E2 -1162.354} C_VEL
LIN {X 0,Y 594.282,Z 462.828,A -85,B 0,C 180,E1 -1163.411,E2 -1163.411} C_VEL
LIN {X 0,Y 594.289,Z 469.675,A -85,B 0,C 180,E1 -1164.57,E2 -1164.57} C_VEL
LIN {X 0,Y 594.27,Z 474.367,A -85,B 0,C 180,E1 -1165.59,E2 -1165.59} C_VEL
LIN {X 0,Y 594.267,Z 477.953,A -85,B 0,C 180,E1 -1166.609,E2 -1166.609} C_VEL
LIN {X 0,Y 594.226,Z 479.806,A -85,B 0,C 180,E1 -1167.287,E2 -1167.287} C_VEL
LIN {X 0,Y 594.24,Z 481.199,A -85,B 0,C 180,E1 -1167.966,E2 -1167.966} C_VEL
LIN {X 0,Y 594.239,Z 482.783,A -85,B 0,C 180,E1 -1169.321,E2 -1169.321} C_VEL
LIN {X 0,Y 594.236,Z 483,A -85,B 0,C 180,E1 -1169.999,E2 -1169.999} C_VEL
LIN {X 0,Y 594.247,Z 482.186,A -85,B 0,C 180,E1 -1171.354,E2 -1171.354} C_VEL
LIN {X 0,Y 594.24,Z 481.203,A -85,B 0,C 180,E1 -1172.032,E2 -1172.032} C_VEL
LIN {X 0,Y 594.226,Z 479.813,A -85,B 0,C 180,E1 -1172.71,E2 -1172.71} C_VEL
LIN {X 0,Y 594.289,Z 476.9,A -85,B 0,C 180,E1 -1173.728,E2 -1173.728} C_VEL
LIN {X 0,Y 594.241,Z 472.955,A -85,B 0,C 180,E1 -1174.748,E2 -1174.748} C_VEL
LIN {X 0,Y 594.304,Z 466.885,A -85,B 0,C 180,E1 -1175.938,E2 -1175.938} C_VEL
LIN {X 0,Y 594.308,Z 460.245,A -85,B 0,C 180,E1 -1176.961,E2 -1176.961} C_VEL
LIN {X 0,Y 594.359,Z 452.001,A -85,B 0,C 180,E1 -1177.985,E2 -1177.985} C_VEL
LIN {X 0,Y 594.404,Z 441.615,A -85,B 0,C 180,E1 -1179.012,E2 -1179.012} C_VEL
LIN {X 0,Y 594.444,Z 430.766,A -85,B 0,C 180,E1 -1179.87,E2 -1179.87} C_VEL
LIN {X 0,Y 594.508,Z 419.802,A -85,B 0,C 180,E1 -1180.557,E2 -1180.557} C_VEL
LIN {X 0,Y 594.601,Z 407.179,A -85,B 0,C 180,E1 -1181.174,E2 -1181.174} C_VEL
LIN {X 0,Y 594.621,Z 395.915,A -85,B 0,C 180,E1 -1181.59,E2 -1181.59} C_VEL
LIN {X 0,Y 594.661,Z 383.579,A -85,B 0,C 180,E1 -1181.913,E2 -1181.913} C_VEL
LIN {X 0,Y 594.695,Z 367.844,A -85,B 0,C 180,E1 -1182.151,E2 -1182.151} C_VEL
LIN {X 0,Y 594.656,Z 273.044,A -85,B 0,C 180,E1 -1183.301,E2 -1183.301} C_VEL
LIN {X 0,Y 594.424,Z 271.017,A -85,B 0,C 180,E1 -1183.372,E2 -1183.372} C_VEL
LIN {X 0,Y 594.489,Z 251.926,A -85,B 0,C 180,E1 -1186.128,E2 -1186.128} C_VEL
LIN {X 0,Y 594.593,Z 233.26,A -85,B 0,C 180,E1 -1188.872,E2 -1188.872} C_VEL
LIN {X 0,Y 594.698,Z 215.728,A -85,B 0,C 180,E1 -1191.489,E2 -1191.489} C_VEL
LIN {X 0,Y 594.378,Z 213.027,A -85,B 0,C 180,E1 -1191.957,E2 -1191.957} C_VEL
LIN {X 0,Y 594.368,Z 212.943,A -85,B 0,C 180,E1 -1194.445,E2 -1194.445} C_VEL
LIN {X 0,Y 594.385,Z 212.94,A -85,B 0,C 180,E1 -1196.698,E2 -1196.698} C_VEL
LIN {X 0,Y 594.375,Z 212.941,A -85,B 0,C 180,E1 -1198.997,E2 -1198.997} C_VEL
LIN {X 0,Y 594.389,Z 212.946,A -85,B 0,C 180,E1 -1201.642,E2 -1201.642} C_VEL
LIN {X 0,Y 594.367,Z 212.943,A -85,B 0,C 180,E1 -1204.579,E2 -1204.579} C_VEL
LIN {X 0,Y 594.386,Z 212.943,A -85,B 0,C 180,E1 -1207.606,E2 -1207.606} C_VEL
LIN {X 0,Y 594.357,Z 212.945,A -85,B 0,C 180,E1 -1210.566,E2 -1210.566} C_VEL
LIN {X 0,Y 594.342,Z 212.945,A -85,B 0,C 180,E1 -1213.299,E2 -1213.299} C_VEL
LIN {X 0,Y 594.343,Z 212.955,A -85,B 0,C 180,E1 -1216.161,E2 -1216.161} C_VEL
LIN {X 0,Y 594.367,Z 212.948,A -85,B 0,C 180,E1 -1218.533,E2 -1218.533} C_VEL
LIN {X 0,Y 594.36,Z 212.942,A -85,B 0,C 180,E1 -1221.296,E2 -1221.296} C_VEL
LIN {X 0,Y 594.34,Z 212.946,A -85,B 0,C 180,E1 -1223.752,E2 -1223.752} C_VEL
LIN {X 0,Y 594.37,Z 212.948,A -85,B 0,C 180,E1 -1226.236,E2 -1226.236} C_VEL
LIN {X 0,Y 594.355,Z 212.951,A -85,B 0,C 180,E1 -1228.646,E2 -1228.646} C_VEL
LIN {X 0,Y 594.335,Z 212.949,A -85,B 0,C 180,E1 -1231.047,E2 -1231.047} C_VEL
LIN {X 0,Y 594.346,Z 212.945,A -85,B 0,C 180,E1 -1233.296,E2 -1233.296} C_VEL
LIN {X 0,Y 594.324,Z 212.947,A -85,B 0,C 180,E1 -1235.576,E2 -1235.576} C_VEL
LIN {X 0,Y 594.334,Z 212.952,A -85,B 0,C 180,E1 -1238.492,E2 -1238.492} C_VEL
LIN {X 0,Y 594.33,Z 212.948,A -85,B 0,C 180,E1 -1241.377,E2 -1241.377} C_VEL
LIN {X 0,Y 594.318,Z 212.948,A -85,B 0,C 180,E1 -1244.214,E2 -1244.214} C_VEL
LIN {X 0,Y 594.313,Z 212.958,A -85,B 0,C 180,E1 -1247.012,E2 -1247.012} C_VEL
LIN {X 0,Y 594.357,Z 212.952,A -85,B 0,C 180,E1 -1249.091,E2 -1249.091} C_VEL
LIN {X 0,Y 594.325,Z 212.947,A -85,B 0,C 180,E1 -1251.838,E2 -1251.838} C_VEL
LIN {X 0,Y 594.313,Z 212.948,A -85,B 0,C 180,E1 -1253.886,E2 -1253.886} C_VEL
LIN {X 0,Y 594.308,Z 212.949,A -85,B 0,C 180,E1 -1255.927,E2 -1255.927} C_VEL
LIN {X 0,Y 594.351,Z 212.944,A -85,B 0,C 180,E1 -1257.963,E2 -1257.963} C_VEL
LIN {X 0,Y 594.373,Z 212.941,A -85,B 0,C 180,E1 -1259.996,E2 -1259.996} C_VEL
LIN {X 0,Y 594.365,Z 212.943,A -85,B 0,C 180,E1 -1262.706,E2 -1262.706} C_VEL
LIN {X 0,Y 594.384,Z 212.95,A -85,B 0,C 180,E1 -1265.423,E2 -1265.423} C_VEL
LIN {X 0,Y 594.391,Z 212.94,A -85,B 0,C 180,E1 -1268.152,E2 -1268.152} C_VEL
LIN {X 0,Y 594.352,Z 212.946,A -85,B 0,C 180,E1 -1271.065,E2 -1271.065} C_VEL
LIN {X 0,Y 594.367,Z 212.951,A -85,B 0,C 180,E1 -1273.674,E2 -1273.674} C_VEL
LIN {X 0,Y 594.341,Z 212.948,A -85,B 0,C 180,E1 -1275.297,E2 -1275.297} C_VEL
LIN {X 0,Y 593.68,Z 213.036,A -85,B 0,C 180,E1 -1275.863,E2 -1275.863} C_VEL
LIN {X 0,Y 590.831,Z 213.392,A -85,B 0,C 180,E1 -1276.781,E2 -1276.781} C_VEL
LIN {X 0,Y 588.421,Z 213.691,A -85,B 0,C 180,E1 -1277.52,E2 -1277.52} C_VEL
LIN {X 0,Y 587.385,Z 213.816,A -85,B 0,C 180,E1 -1278.09,E2 -1278.09} C_VEL
LIN {X 0,Y 587.301,Z 213.824,A -85,B 0,C 180,E1 -1278.283,E2 -1278.283} C_VEL
LIN {X 0,Y 587.32,Z 213.82,A -85,B 0,C 180,E1 -1281.04,E2 -1281.04} C_VEL
LIN {X 0,Y 587.346,Z 213.819,A -85,B 0,C 180,E1 -1283.251,E2 -1283.251} C_VEL
LIN {X 0,Y 587.367,Z 213.969,A -85,B 0,C 180,E1 -1285.556,E2 -1285.556} C_VEL
LIN {X 0,Y 587.623,Z 218.023,A -85,B 0,C 180,E1 -1286.258,E2 -1286.258} C_VEL
LIN {X 0,Y 587.464,Z 235.74,A -85,B 0,C 180,E1 -1289.157,E2 -1289.157} C_VEL
LIN {X 0,Y 587.367,Z 254.17,A -85,B 0,C 180,E1 -1292.13,E2 -1292.13} C_VEL
LIN {X 0,Y 587.405,Z 256.974,A -85,B 0,C 180,E1 -1292.539,E2 -1292.539} C_VEL
LIN {X 0,Y 587.829,Z 261.739,A -85,B 0,C 180,E1 -1292.632,E2 -1292.632} C_VEL
LIN {X 0,Y 587.731,Z 364.809,A -85,B 0,C 180,E1 -1293.916,E2 -1293.916} C_VEL
LIN {X 0,Y 587.679,Z 378.352,A -85,B 0,C 180,E1 -1294.238,E2 -1294.238} C_VEL
LIN {X 0,Y 587.621,Z 390.997,A -85,B 0,C 180,E1 -1294.687,E2 -1294.687} C_VEL
LIN {X 0,Y 587.523,Z 403.863,A -85,B 0,C 180,E1 -1295.309,E2 -1295.309} C_VEL
LIN {X 0,Y 587.466,Z 414.7,A -85,B 0,C 180,E1 -1295.985,E2 -1295.985} C_VEL
LIN {X 0,Y 587.384,Z 425.685,A -85,B 0,C 180,E1 -1296.843,E2 -1296.843} C_VEL
LIN {X 0,Y 587.328,Z 434.719,A -85,B 0,C 180,E1 -1297.719,E2 -1297.719} C_VEL
LIN {X 0,Y 587.258,Z 443.106,A -85,B 0,C 180,E1 -1298.706,E2 -1298.706} C_VEL
LIN {X 0,Y 587.225,Z 449.778,A -85,B 0,C 180,E1 -1299.682,E2 -1299.682} C_VEL
LIN {X 0,Y 587.172,Z 455.225,A -85,B 0,C 180,E1 -1300.658,E2 -1300.658} C_VEL
LIN {X 0,Y 587.175,Z 459.516,A -85,B 0,C 180,E1 -1301.618,E2 -1301.618} C_VEL
LIN {X 0,Y 587.169,Z 462.744,A -85,B 0,C 180,E1 -1302.542,E2 -1302.542} C_VEL
LIN {X 0,Y 587.159,Z 464.298,A -85,B 0,C 180,E1 -1303.105,E2 -1303.105} C_VEL
LIN {X 0,Y 587.142,Z 466.384,A -85,B 0,C 180,E1 -1304.097,E2 -1304.097} C_VEL
LIN {X 0,Y 587.138,Z 467.598,A -85,B 0,C 180,E1 -1305.074,E2 -1305.074} C_VEL
LIN {X 0,Y 587.122,Z 468,A -85,B 0,C 180,E1 -1306.033,E2 -1306.033} C_VEL
LIN {X 0,Y 587.16,Z 467.621,A -85,B 0,C 180,E1 -1306.982,E2 -1306.982} C_VEL
LIN {X 0,Y 587.161,Z 466.511,A -85,B 0,C 180,E1 -1307.913,E2 -1307.913} C_VEL
LIN {X 0,Y 587.136,Z 464.425,A -85,B 0,C 180,E1 -1308.936,E2 -1308.936} C_VEL
LIN {X 0,Y 587.177,Z 461.305,A -85,B 0,C 180,E1 -1309.986,E2 -1309.986} C_VEL
LIN {X 0,Y 587.193,Z 455.932,A -85,B 0,C 180,E1 -1311.29,E2 -1311.29} C_VEL
LIN {X 0,Y 587.196,Z 449.932,A -85,B 0,C 180,E1 -1312.383,E2 -1312.383} C_VEL
LIN {X 0,Y 587.269,Z 442.301,A -85,B 0,C 180,E1 -1313.487,E2 -1313.487} C_VEL
LIN {X 0,Y 587.331,Z 434.017,A -85,B 0,C 180,E1 -1314.444,E2 -1314.444} C_VEL
LIN {X 0,Y 587.359,Z 424.866,A -85,B 0,C 180,E1 -1315.321,E2 -1315.321} C_VEL
LIN {X 0,Y 587.428,Z 414.832,A -85,B 0,C 180,E1 -1316.097,E2 -1316.097} C_VEL
LIN {X 0,Y 587.5,Z 404.177,A -85,B 0,C 180,E1 -1316.764,E2 -1316.764} C_VEL
LIN {X 0,Y 587.589,Z 391.327,A -85,B 0,C 180,E1 -1317.391,E2 -1317.391} C_VEL
LIN {X 0,Y 587.677,Z 379.825,A -85,B 0,C 180,E1 -1317.806,E2 -1317.806} C_VEL
LIN {X 0,Y 587.723,Z 366.629,A -85,B 0,C 180,E1 -1318.14,E2 -1318.14} C_VEL
LIN {X 0,Y 587.752,Z 345.297,A -85,B 0,C 180,E1 -1318.434,E2 -1318.434} C_VEL
LIN {X 0,Y 587.675,Z 259.057,A -85,B 0,C 180,E1 -1319.495,E2 -1319.495} C_VEL
LIN {X 0,Y 587.357,Z 256.873,A -85,B 0,C 180,E1 -1319.557,E2 -1319.557} C_VEL
LIN {X 0,Y 587.469,Z 239.834,A -85,B 0,C 180,E1 -1322.268,E2 -1322.268} C_VEL
LIN {X 0,Y 587.54,Z 223.854,A -85,B 0,C 180,E1 -1324.874,E2 -1324.874} C_VEL
LIN {X 0,Y 587.508,Z 214.757,A -85,B 0,C 180,E1 -1326.377,E2 -1326.377} C_VEL
LIN {X 0,Y 587.334,Z 213.918,A -85,B 0,C 180,E1 -1326.557,E2 -1326.557} C_VEL
LIN {X 0,Y 587.285,Z 213.826,A -85,B 0,C 180,E1 -1328.962,E2 -1328.962} C_VEL
LIN {X 0,Y 587.27,Z 213.829,A -85,B 0,C 180,E1 -1331.873,E2 -1331.873} C_VEL
LIN {X 0,Y 587.294,Z 213.829,A -85,B 0,C 180,E1 -1334.737,E2 -1334.737} C_VEL
LIN {X 0,Y 587.265,Z 213.832,A -85,B 0,C 180,E1 -1336.859,E2 -1336.859} C_VEL
LIN {X 0,Y 587.28,Z 213.824,A -85,B 0,C 180,E1 -1339.66,E2 -1339.66} C_VEL
LIN {X 0,Y 587.314,Z 213.825,A -85,B 0,C 180,E1 -1342.438,E2 -1342.438} C_VEL
LIN {X 0,Y 587.31,Z 213.825,A -85,B 0,C 180,E1 -1345.196,E2 -1345.196} C_VEL
LIN {X 0,Y 587.286,Z 213.823,A -85,B 0,C 180,E1 -1347.944,E2 -1347.944} C_VEL
LIN {X 0,Y 587.333,Z 213.822,A -85,B 0,C 180,E1 -1350.687,E2 -1350.687} C_VEL
LIN {X 0,Y 587.3,Z 213.827,A -85,B 0,C 180,E1 -1353.431,E2 -1353.431} C_VEL
LIN {X 0,Y 587.33,Z 213.823,A -85,B 0,C 180,E1 -1355.494,E2 -1355.494} C_VEL
LIN {X 0,Y 587.299,Z 213.821,A -85,B 0,C 180,E1 -1358.257,E2 -1358.257} C_VEL
LIN {X 0,Y 587.332,Z 213.825,A -85,B 0,C 180,E1 -1361.168,E2 -1361.168} C_VEL
LIN {X 0,Y 587.306,Z 213.821,A -85,B 0,C 180,E1 -1364.271,E2 -1364.271} C_VEL
LIN {X 0,Y 587.297,Z 213.829,A -85,B 0,C 180,E1 -1367.409,E2 -1367.409} C_VEL
LIN {X 0,Y 587.268,Z 213.827,A -85,B 0,C 180,E1 -1370.308,E2 -1370.308} C_VEL
LIN {X 0,Y 587.266,Z 213.828,A -85,B 0,C 180,E1 -1373.262,E2 -1373.262} C_VEL
LIN {X 0,Y 587.29,Z 213.827,A -85,B 0,C 180,E1 -1375.52,E2 -1375.52} C_VEL
LIN {X 0,Y 587.286,Z 213.832,A -85,B 0,C 180,E1 -1377.822,E2 -1377.822} C_VEL
LIN {X 0,Y 587.31,Z 213.823,A -85,B 0,C 180,E1 -1380.521,E2 -1380.521} C_VEL
LIN {X 0,Y 587.284,Z 213.824,A -85,B 0,C 180,E1 -1383.401,E2 -1383.401} C_VEL
LIN {X 0,Y 587.303,Z 213.826,A -85,B 0,C 180,E1 -1385.9,E2 -1385.9} C_VEL
LIN {X 0,Y 587.284,Z 213.831,A -85,B 0,C 180,E1 -1388.484,E2 -1388.484} C_VEL
LIN {X 0,Y 587.311,Z 213.821,A -85,B 0,C 180,E1 -1391.16,E2 -1391.16} C_VEL
LIN {X 0,Y 587.277,Z 213.829,A -85,B 0,C 180,E1 -1394.119,E2 -1394.119} C_VEL
LIN {X 0,Y 587.279,Z 213.828,A -85,B 0,C 180,E1 -1397,E2 -1397} C_VEL
LIN {X 0,Y 587.279,Z 213.824,A -85,B 0,C 180,E1 -1399.752,E2 -1399.752} C_VEL
LIN {X 0,Y 587.31,Z 213.824,A -85,B 0,C 180,E1 -1402.398,E2 -1402.398} C_VEL
LIN {X 0,Y 587.32,Z 213.829,A -85,B 0,C 180,E1 -1404.952,E2 -1404.952} C_VEL
LIN {X 0,Y 587.308,Z 213.824,A -85,B 0,C 180,E1 -1407.427,E2 -1407.427} C_VEL
LIN {X 0,Y 587.291,Z 213.823,A -85,B 0,C 180,E1 -1409.835,E2 -1409.835} C_VEL
LIN {X 0,Y 587.307,Z 213.821,A -85,B 0,C 180,E1 -1412.317,E2 -1412.317} C_VEL
LIN {X 0,Y 587.325,Z 213.83,A -85,B 0,C 180,E1 -1415.247,E2 -1415.247} C_VEL
LIN {X 0,Y 587.303,Z 213.821,A -85,B 0,C 180,E1 -1418.231,E2 -1418.231} C_VEL
LIN {X 0,Y 587.336,Z 213.823,A -85,B 0,C 180,E1 -1421.157,E2 -1421.157} C_VEL
LIN {X 0,Y 587.303,Z 213.824,A -85,B 0,C 180,E1 -1424.03,E2 -1424.03} C_VEL
LIN {X 0,Y 587.342,Z 213.818,A -85,B 0,C 180,E1 -1426.159,E2 -1426.159} C_VEL
LIN {X 0,Y 587.331,Z 213.818,A -85,B 0,C 180,E1 -1428.968,E2 -1428.968} C_VEL
LIN {X 0,Y 587.357,Z 213.825,A -85,B 0,C 180,E1 -1431.75,E2 -1431.75} C_VEL
LIN {X 0,Y 587.343,Z 213.818,A -85,B 0,C 180,E1 -1434.512,E2 -1434.512} C_VEL
LIN {X 0,Y 587.346,Z 213.817,A -85,B 0,C 180,E1 -1437.261,E2 -1437.261} C_VEL
LIN {X 0,Y 587.38,Z 213.822,A -85,B 0,C 180,E1 -1440.005,E2 -1440.005} C_VEL
LIN {X 0,Y 587.369,Z 213.815,A -85,B 0,C 180,E1 -1442.748,E2 -1442.748} C_VEL
LIN {X 0,Y 587.331,Z 213.818,A -85,B 0,C 180,E1 -1445.497,E2 -1445.497} C_VEL
LIN {X 0,Y 587.326,Z 213.828,A -85,B 0,C 180,E1 -1448.26,E2 -1448.26} C_VEL
LIN {X 0,Y 587.361,Z 213.815,A -85,B 0,C 180,E1 -1451.137,E2 -1451.137} C_VEL
LIN {X 0,Y 587.334,Z 213.823,A -85,B 0,C 180,E1 -1454.246,E2 -1454.246} C_VEL
LIN {X 0,Y 587.346,Z 213.824,A -85,B 0,C 180,E1 -1456.812,E2 -1456.812} C_VEL
LIN {X 0,Y 587.312,Z 213.82,A -85,B 0,C 180,E1 -1459.579,E2 -1459.579} C_VEL
LIN {X 0,Y 587.319,Z 213.819,A -85,B 0,C 180,E1 -1461.778,E2 -1461.778} C_VEL
LIN {X 0,Y 587.313,Z 213.828,A -85,B 0,C 180,E1 -1464.763,E2 -1464.763} C_VEL
LIN {X 0,Y 587.312,Z 213.821,A -85,B 0,C 180,E1 -1467.684,E2 -1467.684} C_VEL
LIN {X 0,Y 587.326,Z 213.818,A -85,B 0,C 180,E1 -1470.173,E2 -1470.173} C_VEL
LIN {X 0,Y 587.34,Z 213.818,A -85,B 0,C 180,E1 -1472.582,E2 -1472.582} C_VEL
LIN {X 0,Y 587.314,Z 213.827,A -85,B 0,C 180,E1 -1475.059,E2 -1475.059} C_VEL
LIN {X 0,Y 587.345,Z 213.819,A -85,B 0,C 180,E1 -1477.838,E2 -1477.838} C_VEL
LIN {X 0,Y 587.318,Z 213.819,A -85,B 0,C 180,E1 -1480.257,E2 -1480.257} C_VEL
LIN {X 0,Y 587.3,Z 213.825,A -85,B 0,C 180,E1 -1483.116,E2 -1483.116} C_VEL
LIN {X 0,Y 587.313,Z 213.824,A -85,B 0,C 180,E1 -1486.048,E2 -1486.048} C_VEL
LIN {X 0,Y 587.321,Z 213.819,A -85,B 0,C 180,E1 -1488.929,E2 -1488.929} C_VEL
LIN {X 0,Y 587.329,Z 213.824,A -85,B 0,C 180,E1 -1491.52,E2 -1491.52} C_VEL
LIN {X 0,Y 587.29,Z 213.83,A -85,B 0,C 180,E1 -1494.099,E2 -1494.099} C_VEL
LIN {X 0,Y 587.346,Z 213.816,A -85,B 0,C 180,E1 -1496.889,E2 -1496.889} C_VEL
LIN {X 0,Y 587.331,Z 213.819,A -85,B 0,C 180,E1 -1499.493,E2 -1499.493} C_VEL
LIN {X 0,Y 587.353,Z 213.825,A -85,B 0,C 180,E1 -1502.309,E2 -1502.309} C_VEL
LIN {X 0,Y 587.315,Z 213.821,A -85,B 0,C 180,E1 -1505.239,E2 -1505.239} C_VEL
LIN {X 0,Y 587.361,Z 214.026,A -85,B 0,C 180,E1 -1507.949,E2 -1507.949} C_VEL
LIN {X 0,Y 587.759,Z 218.127,A -85,B 0,C 180,E1 -1508.611,E2 -1508.611} C_VEL
LIN {X 0,Y 587.588,Z 238.637,A -85,B 0,C 180,E1 -1511.7,E2 -1511.7} C_VEL
LIN {X 0,Y 587.453,Z 256.736,A -85,B 0,C 180,E1 -1514.384,E2 -1514.384} C_VEL
LIN {X 0,Y 587.407,Z 271.275,A -85,B 0,C 180,E1 -1516.485,E2 -1516.485} C_VEL
LIN {X 0,Y 587.868,Z 274.637,A -85,B 0,C 180,E1 -1516.562,E2 -1516.562} C_VEL
LIN {X 0,Y 587.752,Z 378.893,A -85,B 0,C 180,E1 -1517.855,E2 -1517.855} C_VEL
LIN {X 0,Y 587.687,Z 392.183,A -85,B 0,C 180,E1 -1518.16,E2 -1518.16} C_VEL
LIN {X 0,Y 587.606,Z 404.77,A -85,B 0,C 180,E1 -1518.59,E2 -1518.59} C_VEL
LIN {X 0,Y 587.556,Z 416.611,A -85,B 0,C 180,E1 -1519.14,E2 -1519.14} C_VEL
LIN {X 0,Y 587.438,Z 428.187,A -85,B 0,C 180,E1 -1519.835,E2 -1519.835} C_VEL
LIN {X 0,Y 587.393,Z 438.586,A -85,B 0,C 180,E1 -1520.617,E2 -1520.617} C_VEL
LIN {X 0,Y 587.3,Z 447.036,A -85,B 0,C 180,E1 -1521.396,E2 -1521.396} C_VEL
LIN {X 0,Y 587.275,Z 454.952,A -85,B 0,C 180,E1 -1522.262,E2 -1522.262} C_VEL
LIN {X 0,Y 587.233,Z 461.461,A -85,B 0,C 180,E1 -1523.125,E2 -1523.125} C_VEL
LIN {X 0,Y 587.237,Z 467.861,A -85,B 0,C 180,E1 -1524.16,E2 -1524.16} C_VEL
LIN {X 0,Y 587.147,Z 472.945,A -85,B 0,C 180,E1 -1525.193,E2 -1525.193} C_VEL
LIN {X 0,Y 587.213,Z 476.892,A -85,B 0,C 180,E1 -1526.225,E2 -1526.225} C_VEL
LIN {X 0,Y 587.132,Z 479.806,A -85,B 0,C 180,E1 -1527.254,E2 -1527.254} C_VEL
LIN {X 0,Y 587.139,Z 481.198,A -85,B 0,C 180,E1 -1527.941,E2 -1527.941} C_VEL
LIN {X 0,Y 587.14,Z 482.784,A -85,B 0,C 180,E1 -1529.313,E2 -1529.313} C_VEL
LIN {X 0,Y 587.137,Z 483,A -85,B 0,C 180,E1 -1529.999,E2 -1529.999} C_VEL
LIN {X 0,Y 587.147,Z 482.187,A -85,B 0,C 180,E1 -1531.371,E2 -1531.371} C_VEL
LIN {X 0,Y 587.139,Z 481.203,A -85,B 0,C 180,E1 -1532.057,E2 -1532.057} C_VEL
LIN {X 0,Y 587.132,Z 479.813,A -85,B 0,C 180,E1 -1532.743,E2 -1532.743} C_VEL
LIN {X 0,Y 587.213,Z 476.9,A -85,B 0,C 180,E1 -1533.773,E2 -1533.773} C_VEL
LIN {X 0,Y 587.147,Z 472.954,A -85,B 0,C 180,E1 -1534.805,E2 -1534.805} C_VEL
LIN {X 0,Y 587.217,Z 466.885,A -85,B 0,C 180,E1 -1536.01,E2 -1536.01} C_VEL
LIN {X 0,Y 587.246,Z 460.246,A -85,B 0,C 180,E1 -1537.045,E2 -1537.045} C_VEL
LIN {X 0,Y 587.297,Z 452.001,A -85,B 0,C 180,E1 -1538.082,E2 -1538.082} C_VEL
LIN {X 0,Y 587.357,Z 441.616,A -85,B 0,C 180,E1 -1539.121,E2 -1539.121} C_VEL
LIN {X 0,Y 587.44,Z 430.766,A -85,B 0,C 180,E1 -1539.989,E2 -1539.989} C_VEL
LIN {X 0,Y 587.524,Z 419.805,A -85,B 0,C 180,E1 -1540.684,E2 -1540.684} C_VEL
LIN {X 0,Y 587.618,Z 408.222,A -85,B 0,C 180,E1 -1541.263,E2 -1541.263} C_VEL
LIN {X 0,Y 587.686,Z 395.913,A -85,B 0,C 180,E1 -1541.729,E2 -1541.729} C_VEL
LIN {X 0,Y 587.714,Z 383.577,A -85,B 0,C 180,E1 -1542.056,E2 -1542.056} C_VEL
LIN {X 0,Y 587.768,Z 367.844,A -85,B 0,C 180,E1 -1542.296,E2 -1542.296} C_VEL
LIN {X 0,Y 587.685,Z 273.165,A -85,B 0,C 180,E1 -1543.46,E2 -1543.46} C_VEL
LIN {X 0,Y 587.383,Z 271.292,A -85,B 0,C 180,E1 -1543.513,E2 -1543.513} C_VEL
LIN {X 0,Y 587.476,Z 255.546,A -85,B 0,C 180,E1 -1545.791,E2 -1545.791} C_VEL
LIN {X 0,Y 587.588,Z 237.447,A -85,B 0,C 180,E1 -1548.478,E2 -1548.478} C_VEL
LIN {X 0,Y 587.724,Z 219.81,A -85,B 0,C 180,E1 -1551.135,E2 -1551.135} C_VEL
LIN {X 0,Y 587.46,Z 214.534,A -85,B 0,C 180,E1 -1551.952,E2 -1551.952} C_VEL
LIN {X 0,Y 587.321,Z 213.877,A -85,B 0,C 180,E1 -1552.142,E2 -1552.142} C_VEL
LIN {X 0,Y 587.316,Z 213.821,A -85,B 0,C 180,E1 -1554.758,E2 -1554.758} C_VEL
LIN {X 0,Y 587.331,Z 213.82,A -85,B 0,C 180,E1 -1557.044,E2 -1557.044} C_VEL
LIN {X 0,Y 587.317,Z 213.824,A -85,B 0,C 180,E1 -1559.379,E2 -1559.379} C_VEL
LIN {X 0,Y 587.349,Z 213.827,A -85,B 0,C 180,E1 -1561.834,E2 -1561.834} C_VEL
LIN {X 0,Y 587.339,Z 213.821,A -85,B 0,C 180,E1 -1564.344,E2 -1564.344} C_VEL
LIN {X 0,Y 587.341,Z 213.821,A -85,B 0,C 180,E1 -1567.606,E2 -1567.606} C_VEL
LIN {X 0,Y 587.306,Z 213.829,A -85,B 0,C 180,E1 -1570.253,E2 -1570.253} C_VEL
LIN {X 0,Y 587.285,Z 213.824,A -85,B 0,C 180,E1 -1573.007,E2 -1573.007} C_VEL
LIN {X 0,Y 587.302,Z 213.827,A -85,B 0,C 180,E1 -1575.887,E2 -1575.887} C_VEL
LIN {X 0,Y 587.306,Z 213.822,A -85,B 0,C 180,E1 -1578.926,E2 -1578.926} C_VEL
LIN {X 0,Y 587.308,Z 213.821,A -85,B 0,C 180,E1 -1581.516,E2 -1581.516} C_VEL
LIN {X 0,Y 587.275,Z 213.83,A -85,B 0,C 180,E1 -1584.096,E2 -1584.096} C_VEL
LIN {X 0,Y 587.33,Z 213.822,A -85,B 0,C 180,E1 -1586.886,E2 -1586.886} C_VEL
LIN {X 0,Y 587.309,Z 213.82,A -85,B 0,C 180,E1 -1589.491,E2 -1589.491} C_VEL
LIN {X 0,Y 587.29,Z 213.829,A -85,B 0,C 180,E1 -1592.315,E2 -1592.315} C_VEL
LIN {X 0,Y 587.291,Z 213.825,A -85,B 0,C 180,E1 -1595.236,E2 -1595.236} C_VEL
LIN {X 0,Y 587.282,Z 213.826,A -85,B 0,C 180,E1 -1598.221,E2 -1598.221} C_VEL
LIN {X 0,Y 587.313,Z 213.825,A -85,B 0,C 180,E1 -1601.147,E2 -1601.147} C_VEL
LIN {X 0,Y 587.271,Z 213.825,A -85,B 0,C 180,E1 -1604.02,E2 -1604.02} C_VEL
LIN {X 0,Y 587.305,Z 213.822,A -85,B 0,C 180,E1 -1606.149,E2 -1606.149} C_VEL
LIN {X 0,Y 587.325,Z 213.829,A -85,B 0,C 180,E1 -1608.958,E2 -1608.958} C_VEL
LIN {X 0,Y 587.295,Z 213.823,A -85,B 0,C 180,E1 -1611.74,E2 -1611.74} C_VEL
LIN {X 0,Y 587.273,Z 213.826,A -85,B 0,C 180,E1 -1613.813,E2 -1613.813} C_VEL
LIN {X 0,Y 587.265,Z 213.827,A -85,B 0,C 180,E1 -1615.878,E2 -1615.878} C_VEL
LIN {X 0,Y 587.325,Z 213.819,A -85,B 0,C 180,E1 -1617.938,E2 -1617.938} C_VEL
LIN {X 0,Y 587.344,Z 213.817,A -85,B 0,C 180,E1 -1619.995,E2 -1619.995} C_VEL
LIN {X 0,Y 587.334,Z 213.819,A -85,B 0,C 180,E1 -1622.739,E2 -1622.739} C_VEL
LIN {X 0,Y 587.348,Z 213.826,A -85,B 0,C 180,E1 -1625.488,E2 -1625.488} C_VEL
LIN {X 0,Y 587.341,Z 213.817,A -85,B 0,C 180,E1 -1628.25,E2 -1628.25} C_VEL
LIN {X 0,Y 587.32,Z 213.823,A -85,B 0,C 180,E1 -1631.129,E2 -1631.129} C_VEL
LIN {X 0,Y 587.359,Z 213.816,A -85,B 0,C 180,E1 -1634.266,E2 -1634.266} C_VEL
LIN {X 0,Y 587.332,Z 213.824,A -85,B 0,C 180,E1 -1637.401,E2 -1637.401} C_VEL
LIN {X 0,Y 587.301,Z 213.824,A -85,B 0,C 180,E1 -1638.283,E2 -1638.283} C_VEL
LIN {X 0,Y 586.639,Z 213.907,A -85,B 0,C 180,E1 -1638.855,E2 -1638.855} C_VEL
LIN {X 0,Y 583.802,Z 214.268,A -85,B 0,C 180,E1 -1639.783,E2 -1639.783} C_VEL
LIN {X 0,Y 581.396,Z 214.566,A -85,B 0,C 180,E1 -1640.53,E2 -1640.53} C_VEL
LIN {X 0,Y 580.351,Z 214.692,A -85,B 0,C 180,E1 -1641.107,E2 -1641.107} C_VEL
LIN {X 0,Y 580.259,Z 214.703,A -85,B 0,C 180,E1 -1641.302,E2 -1641.302} C_VEL
LIN {X 0,Y 580.279,Z 214.703,A -85,B 0,C 180,E1 -1643.551,E2 -1643.551} C_VEL
LIN {X 0,Y 580.311,Z 214.894,A -85,B 0,C 180,E1 -1645.456,E2 -1645.456} C_VEL
LIN {X 0,Y 580.664,Z 218.635,A -85,B 0,C 180,E1 -1646.113,E2 -1646.113} C_VEL
LIN {X 0,Y 580.444,Z 236.966,A -85,B 0,C 180,E1 -1649.149,E2 -1649.149} C_VEL
LIN {X 0,Y 580.324,Z 253.643,A -85,B 0,C 180,E1 -1651.872,E2 -1651.872} C_VEL
LIN {X 0,Y 580.372,Z 256.907,A -85,B 0,C 180,E1 -1652.368,E2 -1652.368} C_VEL
LIN {X 0,Y 580.919,Z 261.119,A -85,B 0,C 180,E1 -1652.462,E2 -1652.462} C_VEL
LIN {X 0,Y 580.83,Z 363.552,A -85,B 0,C 180,E1 -1653.75,E2 -1653.75} C_VEL
LIN {X 0,Y 580.72,Z 376.569,A -85,B 0,C 180,E1 -1654.042,E2 -1654.042} C_VEL
LIN {X 0,Y 580.66,Z 388.576,A -85,B 0,C 180,E1 -1654.452,E2 -1654.452} C_VEL
LIN {X 0,Y 580.568,Z 400.324,A -85,B 0,C 180,E1 -1654.986,E2 -1654.986} C_VEL
LIN {X 0,Y 580.461,Z 411.16,A -85,B 0,C 180,E1 -1655.621,E2 -1655.621} C_VEL
LIN {X 0,Y 580.379,Z 421.643,A -85,B 0,C 180,E1 -1656.387,E2 -1656.387} C_VEL
LIN {X 0,Y 580.29,Z 431.293,A -85,B 0,C 180,E1 -1657.26,E2 -1657.26} C_VEL
LIN {X 0,Y 580.214,Z 439.347,A -85,B 0,C 180,E1 -1658.143,E2 -1658.143} C_VEL
LIN {X 0,Y 580.152,Z 447.035,A -85,B 0,C 180,E1 -1659.171,E2 -1659.171} C_VEL
LIN {X 0,Y 580.116,Z 453.474,A -85,B 0,C 180,E1 -1660.253,E2 -1660.253} C_VEL
LIN {X 0,Y 580.111,Z 458.491,A -85,B 0,C 180,E1 -1661.315,E2 -1661.315} C_VEL
LIN {X 0,Y 580.078,Z 462.299,A -85,B 0,C 180,E1 -1662.352,E2 -1662.352} C_VEL
LIN {X 0,Y 580.023,Z 465.659,A -85,B 0,C 180,E1 -1663.672,E2 -1663.672} C_VEL
LIN {X 0,Y 580.039,Z 467.148,A -85,B 0,C 180,E1 -1664.638,E2 -1664.638} C_VEL
LIN {X 0,Y 580.039,Z 467.896,A -85,B 0,C 180,E1 -1665.622,E2 -1665.622} C_VEL
LIN {X 0,Y 580.023,Z 467.838,A -85,B 0,C 180,E1 -1666.625,E2 -1666.625} C_VEL
LIN {X 0,Y 580.05,Z 466.933,A -85,B 0,C 180,E1 -1667.643,E2 -1667.643} C_VEL
LIN {X 0,Y 580.033,Z 465.112,A -85,B 0,C 180,E1 -1668.685,E2 -1668.685} C_VEL
LIN {X 0,Y 580.08,Z 461.24,A -85,B 0,C 180,E1 -1670.052,E2 -1670.052} C_VEL
LIN {X 0,Y 580.104,Z 456.757,A -85,B 0,C 180,E1 -1671.176,E2 -1671.176} C_VEL
LIN {X 0,Y 580.108,Z 450.73,A -85,B 0,C 180,E1 -1672.328,E2 -1672.328} C_VEL
LIN {X 0,Y 580.158,Z 444.124,A -85,B 0,C 180,E1 -1673.332,E2 -1673.332} C_VEL
LIN {X 0,Y 580.25,Z 435.962,A -85,B 0,C 180,E1 -1674.342,E2 -1674.342} C_VEL
LIN {X 0,Y 580.312,Z 426.268,A -85,B 0,C 180,E1 -1675.307,E2 -1675.307} C_VEL
LIN {X 0,Y 580.403,Z 415.793,A -85,B 0,C 180,E1 -1676.153,E2 -1676.153} C_VEL
LIN {X 0,Y 580.494,Z 405.467,A -85,B 0,C 180,E1 -1676.819,E2 -1676.819} C_VEL
LIN {X 0,Y 580.606,Z 394.048,A -85,B 0,C 180,E1 -1677.41,E2 -1677.41} C_VEL
LIN {X 0,Y 580.729,Z 381.743,A -85,B 0,C 180,E1 -1677.887,E2 -1677.887} C_VEL
LIN {X 0,Y 580.804,Z 369.827,A -85,B 0,C 180,E1 -1678.216,E2 -1678.216} C_VEL
LIN {X 0,Y 580.846,Z 356.26,A -85,B 0,C 180,E1 -1678.448,E2 -1678.448} C_VEL
LIN {X 0,Y 580.723,Z 259.526,A -85,B 0,C 180,E1 -1679.653,E2 -1679.653} C_VEL
LIN {X 0,Y 580.352,Z 257.156,A -85,B 0,C 180,E1 -1679.707,E2 -1679.707} C_VEL
LIN {X 0,Y 580.333,Z 254.789,A -85,B 0,C 180,E1 -1680.032,E2 -1680.032} C_VEL
LIN {X 0,Y 580.47,Z 237.794,A -85,B 0,C 180,E1 -1682.805,E2 -1682.805} C_VEL
LIN {X 0,Y 580.609,Z 220.306,A -85,B 0,C 180,E1 -1685.699,E2 -1685.699} C_VEL
LIN {X 0,Y 580.495,Z 215.833,A -85,B 0,C 180,E1 -1686.453,E2 -1686.453} C_VEL
LIN {X 0,Y 580.313,Z 214.781,A -85,B 0,C 180,E1 -1686.675,E2 -1686.675} C_VEL
LIN {X 0,Y 580.218,Z 214.706,A -85,B 0,C 180,E1 -1689.437,E2 -1689.437} C_VEL
LIN {X 0,Y 580.217,Z 214.706,A -85,B 0,C 180,E1 -1691.645,E2 -1691.645} C_VEL
LIN {X 0,Y 580.251,Z 214.71,A -85,B 0,C 180,E1 -1694.548,E2 -1694.548} C_VEL
LIN {X 0,Y 580.223,Z 214.712,A -85,B 0,C 180,E1 -1696.696,E2 -1696.696} C_VEL
LIN {X 0,Y 580.247,Z 214.7,A -85,B 0,C 180,E1 -1699.534,E2 -1699.534} C_VEL
LIN {X 0,Y 580.289,Z 214.699,A -85,B 0,C 180,E1 -1702.345,E2 -1702.345} C_VEL
LIN {X 0,Y 580.282,Z 214.701,A -85,B 0,C 180,E1 -1705.138,E2 -1705.138} C_VEL
LIN {X 0,Y 580.257,Z 214.699,A -85,B 0,C 180,E1 -1707.919,E2 -1707.919} C_VEL
LIN {X 0,Y 580.302,Z 214.698,A -85,B 0,C 180,E1 -1710.695,E2 -1710.695} C_VEL
LIN {X 0,Y 580.249,Z 214.705,A -85,B 0,C 180,E1 -1713.473,E2 -1713.473} C_VEL
LIN {X 0,Y 580.288,Z 214.7,A -85,B 0,C 180,E1 -1715.561,E2 -1715.561} C_VEL
LIN {X 0,Y 580.263,Z 214.698,A -85,B 0,C 180,E1 -1718.358,E2 -1718.358} C_VEL
LIN {X 0,Y 580.304,Z 214.701,A -85,B 0,C 180,E1 -1721.236,E2 -1721.236} C_VEL
LIN {X 0,Y 580.253,Z 214.699,A -85,B 0,C 180,E1 -1724.348,E2 -1724.348} C_VEL
LIN {X 0,Y 580.239,Z 214.702,A -85,B 0,C 180,E1 -1726.918,E2 -1726.918} C_VEL
LIN {X 0,Y 580.242,Z 214.709,A -85,B 0,C 180,E1 -1729.826,E2 -1729.826} C_VEL
LIN {X 0,Y 580.211,Z 214.71,A -85,B 0,C 180,E1 -1732.056,E2 -1732.056} C_VEL
LIN {X 0,Y 580.254,Z 214.7,A -85,B 0,C 180,E1 -1735.083,E2 -1735.083} C_VEL
LIN {X 0,Y 580.256,Z 214.709,A -85,B 0,C 180,E1 -1737.868,E2 -1737.868} C_VEL
LIN {X 0,Y 580.253,Z 214.701,A -85,B 0,C 180,E1 -1740.705,E2 -1740.705} C_VEL
LIN {X 0,Y 580.251,Z 214.7,A -85,B 0,C 180,E1 -1743.323,E2 -1743.323} C_VEL
LIN {X 0,Y 580.271,Z 214.701,A -85,B 0,C 180,E1 -1745.773,E2 -1745.773} C_VEL
LIN {X 0,Y 580.238,Z 214.709,A -85,B 0,C 180,E1 -1748.151,E2 -1748.151} C_VEL
LIN {X 0,Y 580.271,Z 214.7,A -85,B 0,C 180,E1 -1750.847,E2 -1750.847} C_VEL
LIN {X 0,Y 580.234,Z 214.702,A -85,B 0,C 180,E1 -1753.663,E2 -1753.663} C_VEL
LIN {X 0,Y 580.242,Z 214.712,A -85,B 0,C 180,E1 -1756.614,E2 -1756.614} C_VEL
LIN {X 0,Y 580.277,Z 214.699,A -85,B 0,C 180,E1 -1759.164,E2 -1759.164} C_VEL
LIN {X 0,Y 580.252,Z 214.7,A -85,B 0,C 180,E1 -1761.933,E2 -1761.933} C_VEL
LIN {X 0,Y 580.268,Z 214.702,A -85,B 0,C 180,E1 -1764.462,E2 -1764.462} C_VEL
LIN {X 0,Y 580.258,Z 214.709,A -85,B 0,C 180,E1 -1766.981,E2 -1766.981} C_VEL
LIN {X 0,Y 580.266,Z 214.702,A -85,B 0,C 180,E1 -1769.431,E2 -1769.431} C_VEL
LIN {X 0,Y 580.262,Z 214.698,A -85,B 0,C 180,E1 -1772.149,E2 -1772.149} C_VEL
LIN {X 0,Y 580.277,Z 214.702,A -85,B 0,C 180,E1 -1774.926,E2 -1774.926} C_VEL
LIN {X 0,Y 580.26,Z 214.7,A -85,B 0,C 180,E1 -1777.953,E2 -1777.953} C_VEL
LIN {X 0,Y 580.284,Z 214.698,A -85,B 0,C 180,E1 -1780.919,E2 -1780.919} C_VEL
LIN {X 0,Y 580.257,Z 214.704,A -85,B 0,C 180,E1 -1783.831,E2 -1783.831} C_VEL
LIN {X 0,Y 580.312,Z 214.696,A -85,B 0,C 180,E1 -1785.988,E2 -1785.988} C_VEL
LIN {X 0,Y 580.3,Z 214.694,A -85,B 0,C 180,E1 -1788.832,E2 -1788.832} C_VEL
LIN {X 0,Y 580.319,Z 214.7,A -85,B 0,C 180,E1 -1791.649,E2 -1791.649} C_VEL
LIN {X 0,Y 580.312,Z 214.694,A -85,B 0,C 180,E1 -1794.445,E2 -1794.445} C_VEL
LIN {X 0,Y 580.315,Z 214.692,A -85,B 0,C 180,E1 -1797.228,E2 -1797.228} C_VEL
LIN {X 0,Y 580.349,Z 214.698,A -85,B 0,C 180,E1 -1800.005,E2 -1800.005} C_VEL
LIN {X 0,Y 580.333,Z 214.691,A -85,B 0,C 180,E1 -1802.781,E2 -1802.781} C_VEL
LIN {X 0,Y 580.3,Z 214.694,A -85,B 0,C 180,E1 -1805.564,E2 -1805.564} C_VEL
LIN {X 0,Y 580.3,Z 214.705,A -85,B 0,C 180,E1 -1808.361,E2 -1808.361} C_VEL
LIN {X 0,Y 580.313,Z 214.692,A -85,B 0,C 180,E1 -1811.195,E2 -1811.195} C_VEL
LIN {X 0,Y 580.304,Z 214.695,A -85,B 0,C 180,E1 -1814.021,E2 -1814.021} C_VEL
LIN {X 0,Y 580.304,Z 214.699,A -85,B 0,C 180,E1 -1816.909,E2 -1816.909} C_VEL
LIN {X 0,Y 580.287,Z 214.695,A -85,B 0,C 180,E1 -1819.826,E2 -1819.826} C_VEL
LIN {X 0,Y 580.263,Z 214.699,A -85,B 0,C 180,E1 -1822.056,E2 -1822.056} C_VEL
LIN {X 0,Y 580.289,Z 214.703,A -85,B 0,C 180,E1 -1825.084,E2 -1825.084} C_VEL
LIN {X 0,Y 580.258,Z 214.699,A -85,B 0,C 180,E1 -1827.85,E2 -1827.85} C_VEL
LIN {X 0,Y 580.283,Z 214.7,A -85,B 0,C 180,E1 -1830.693,E2 -1830.693} C_VEL
LIN {X 0,Y 580.295,Z 214.703,A -85,B 0,C 180,E1 -1833.314,E2 -1833.314} C_VEL
LIN {X 0,Y 580.242,Z 214.704,A -85,B 0,C 180,E1 -1835.755,E2 -1835.755} C_VEL
LIN {X 0,Y 580.297,Z 214.694,A -85,B 0,C 180,E1 -1838.148,E2 -1838.148} C_VEL
LIN {X 0,Y 580.294,Z 214.696,A -85,B 0,C 180,E1 -1840.846,E2 -1840.846} C_VEL
LIN {X 0,Y 580.251,Z 214.709,A -85,B 0,C 180,E1 -1843.663,E2 -1843.663} C_VEL
LIN {X 0,Y 580.249,Z 214.7,A -85,B 0,C 180,E1 -1846.615,E2 -1846.615} C_VEL
LIN {X 0,Y 580.291,Z 214.697,A -85,B 0,C 180,E1 -1849.155,E2 -1849.155} C_VEL
LIN {X 0,Y 580.299,Z 214.703,A -85,B 0,C 180,E1 -1851.928,E2 -1851.928} C_VEL
LIN {X 0,Y 580.24,Z 214.703,A -85,B 0,C 180,E1 -1854.451,E2 -1854.451} C_VEL
LIN {X 0,Y 580.297,Z 214.694,A -85,B 0,C 180,E1 -1856.975,E2 -1856.975} C_VEL
LIN {X 0,Y 580.293,Z 214.696,A -85,B 0,C 180,E1 -1859.424,E2 -1859.424} C_VEL
LIN {X 0,Y 580.299,Z 214.705,A -85,B 0,C 180,E1 -1862.143,E2 -1862.143} C_VEL
LIN {X 0,Y 580.294,Z 214.698,A -85,B 0,C 180,E1 -1864.919,E2 -1864.919} C_VEL
LIN {X 0,Y 580.315,Z 214.901,A -85,B 0,C 180,E1 -1867.808,E2 -1867.808} C_VEL
LIN {X 0,Y 580.834,Z 219.329,A -85,B 0,C 180,E1 -1868.529,E2 -1868.529} C_VEL
LIN {X 0,Y 580.629,Z 238.637,A -85,B 0,C 180,E1 -1871.473,E2 -1871.473} C_VEL
LIN {X 0,Y 580.476,Z 256.736,A -85,B 0,C 180,E1 -1874.191,E2 -1874.191} C_VEL
LIN {X 0,Y 580.386,Z 271.277,A -85,B 0,C 180,E1 -1876.318,E2 -1876.318} C_VEL
LIN {X 0,Y 580.975,Z 276.426,A -85,B 0,C 180,E1 -1876.422,E2 -1876.422} C_VEL
LIN {X 0,Y 580.826,Z 378.892,A -85,B 0,C 180,E1 -1877.708,E2 -1877.708} C_VEL
LIN {X 0,Y 580.746,Z 392.183,A -85,B 0,C 180,E1 -1878.016,E2 -1878.016} C_VEL
LIN {X 0,Y 580.636,Z 404.348,A -85,B 0,C 180,E1 -1878.435,E2 -1878.435} C_VEL
LIN {X 0,Y 580.563,Z 416.609,A -85,B 0,C 180,E1 -1879.008,E2 -1879.008} C_VEL
LIN {X 0,Y 580.418,Z 428.186,A -85,B 0,C 180,E1 -1879.711,E2 -1879.711} C_VEL
LIN {X 0,Y 580.343,Z 438.587,A -85,B 0,C 180,E1 -1880.502,E2 -1880.502} C_VEL
LIN {X 0,Y 580.264,Z 447.051,A -85,B 0,C 180,E1 -1881.291,E2 -1881.291} C_VEL
LIN {X 0,Y 580.224,Z 454.952,A -85,B 0,C 180,E1 -1882.167,E2 -1882.167} C_VEL
LIN {X 0,Y 580.159,Z 462.637,A -85,B 0,C 180,E1 -1883.22,E2 -1883.22} C_VEL
LIN {X 0,Y 580.14,Z 469.674,A -85,B 0,C 180,E1 -1884.437,E2 -1884.437} C_VEL
LIN {X 0,Y 580.108,Z 474.367,A -85,B 0,C 180,E1 -1885.482,E2 -1885.482} C_VEL
LIN {X 0,Y 580.123,Z 477.954,A -85,B 0,C 180,E1 -1886.526,E2 -1886.526} C_VEL
LIN {X 0,Y 580.043,Z 479.806,A -85,B 0,C 180,E1 -1887.221,E2 -1887.221} C_VEL
LIN {X 0,Y 580.038,Z 481.197,A -85,B 0,C 180,E1 -1887.916,E2 -1887.916} C_VEL
LIN {X 0,Y 580.04,Z 482.784,A -85,B 0,C 180,E1 -1889.305,E2 -1889.305} C_VEL
LIN {X 0,Y 580.037,Z 483,A -85,B 0,C 180,E1 -1889.999,E2 -1889.999} C_VEL
LIN {X 0,Y 580.046,Z 482.187,A -85,B 0,C 180,E1 -1891.387,E2 -1891.387} C_VEL
LIN {X 0,Y 580.038,Z 481.202,A -85,B 0,C 180,E1 -1892.082,E2 -1892.082} C_VEL
LIN {X 0,Y 580.043,Z 479.813,A -85,B 0,C 180,E1 -1892.777,E2 -1892.777} C_VEL
LIN {X 0,Y 580.11,Z 476.9,A -85,B 0,C 180,E1 -1893.819,E2 -1893.819} C_VEL
LIN {X 0,Y 580.053,Z 472.954,A -85,B 0,C 180,E1 -1894.864,E2 -1894.864} C_VEL
LIN {X 0,Y 580.164,Z 467.873,A -85,B 0,C 180,E1 -1895.909,E2 -1895.909} C_VEL
LIN {X 0,Y 580.185,Z 460.247,A -85,B 0,C 180,E1 -1897.131,E2 -1897.131} C_VEL
LIN {X 0,Y 580.246,Z 452.002,A -85,B 0,C 180,E1 -1898.181,E2 -1898.181} C_VEL
LIN {X 0,Y 580.333,Z 441.616,A -85,B 0,C 180,E1 -1899.232,E2 -1899.232} C_VEL
LIN {X 0,Y 580.434,Z 430.765,A -85,B 0,C 180,E1 -1900.11,E2 -1900.11} C_VEL
LIN {X 0,Y 580.537,Z 419.807,A -85,B 0,C 180,E1 -1900.814,E2 -1900.814} C_VEL
LIN {X 0,Y 580.663,Z 407.58,A -85,B 0,C 180,E1 -1901.428,E2 -1901.428} C_VEL
LIN {X 0,Y 580.732,Z 395.911,A -85,B 0,C 180,E1 -1901.871,E2 -1901.871} C_VEL
LIN {X 0,Y 580.786,Z 383.576,A -85,B 0,C 180,E1 -1902.202,E2 -1902.202} C_VEL
LIN {X 0,Y 580.832,Z 367.844,A -85,B 0,C 180,E1 -1902.445,E2 -1902.445} C_VEL
LIN {X 0,Y 580.904,Z 274.833,A -85,B 0,C 180,E1 -1903.6,E2 -1903.6} C_VEL
LIN {X 0,Y 580.386,Z 271.304,A -85,B 0,C 180,E1 -1903.679,E2 -1903.679} C_VEL
LIN {X 0,Y 580.501,Z 253.133,A -85,B 0,C 180,E1 -1906.347,E2 -1906.347} C_VEL
LIN {X 0,Y 580.646,Z 235.034,A -85,B 0,C 180,E1 -1909.073,E2 -1909.073} C_VEL
LIN {X 0,Y 580.817,Z 218.125,A -85,B 0,C 180,E1 -1911.655,E2 -1911.655} C_VEL
LIN {X 0,Y 580.306,Z 214.775,A -85,B 0,C 180,E1 -1912.237,E2 -1912.237} C_VEL
LIN {X 0,Y 580.292,Z 214.698,A -85,B 0,C 180,E1 -1915.079,E2 -1915.079} C_VEL
LIN {X 0,Y 580.295,Z 214.704,A -85,B 0,C 180,E1 -1917.856,E2 -1917.856} C_VEL
LIN {X 0,Y 580.281,Z 214.696,A -85,B 0,C 180,E1 -1920.692,E2 -1920.692} C_VEL
LIN {X 0,Y 580.302,Z 214.696,A -85,B 0,C 180,E1 -1923.314,E2 -1923.314} C_VEL
LIN {X 0,Y 580.242,Z 214.709,A -85,B 0,C 180,E1 -1925.753,E2 -1925.753} C_VEL
LIN {X 0,Y 580.284,Z 214.705,A -85,B 0,C 180,E1 -1928.145,E2 -1928.145} C_VEL
LIN {X 0,Y 580.292,Z 214.695,A -85,B 0,C 180,E1 -1930.842,E2 -1930.842} C_VEL
LIN {X 0,Y 580.236,Z 214.705,A -85,B 0,C 180,E1 -1933.659,E2 -1933.659} C_VEL
LIN {X 0,Y 580.231,Z 214.707,A -85,B 0,C 180,E1 -1936.612,E2 -1936.612} C_VEL
LIN {X 0,Y 580.276,Z 214.697,A -85,B 0,C 180,E1 -1939.152,E2 -1939.152} C_VEL
LIN {X 0,Y 580.277,Z 214.7,A -85,B 0,C 180,E1 -1941.926,E2 -1941.926} C_VEL
LIN {X 0,Y 580.227,Z 214.714,A -85,B 0,C 180,E1 -1944.448,E2 -1944.448} C_VEL
LIN {X 0,Y 580.28,Z 214.699,A -85,B 0,C 180,E1 -1946.972,E2 -1946.972} C_VEL
LIN {X 0,Y 580.271,Z 214.697,A -85,B 0,C 180,E1 -1949.421,E2 -1949.421} C_VEL
LIN {X 0,Y 580.233,Z 214.706,A -85,B 0,C 180,E1 -1952.149,E2 -1952.149} C_VEL
LIN {X 0,Y 580.27,Z 214.704,A -85,B 0,C 180,E1 -1954.915,E2 -1954.915} C_VEL
LIN {X 0,Y 580.217,Z 214.704,A -85,B 0,C 180,E1 -1957.942,E2 -1957.942} C_VEL
LIN {X 0,Y 580.27,Z 214.707,A -85,B 0,C 180,E1 -1960.909,E2 -1960.909} C_VEL
LIN {X 0,Y 580.223,Z 214.703,A -85,B 0,C 180,E1 -1963.82,E2 -1963.82} C_VEL
LIN {X 0,Y 580.263,Z 214.698,A -85,B 0,C 180,E1 -1965.978,E2 -1965.978} C_VEL
LIN {X 0,Y 580.294,Z 214.702,A -85,B 0,C 180,E1 -1968.823,E2 -1968.823} C_VEL
LIN {X 0,Y 580.271,Z 214.699,A -85,B 0,C 180,E1 -1971.639,E2 -1971.639} C_VEL
LIN {X 0,Y 580.236,Z 214.703,A -85,B 0,C 180,E1 -1973.738,E2 -1973.738} C_VEL
LIN {X 0,Y 580.224,Z 214.705,A -85,B 0,C 180,E1 -1975.828,E2 -1975.828} C_VEL
LIN {X 0,Y 580.299,Z 214.695,A -85,B 0,C 180,E1 -1977.913,E2 -1977.913} C_VEL
LIN {X 0,Y 580.315,Z 214.692,A -85,B 0,C 180,E1 -1979.995,E2 -1979.995} C_VEL
LIN {X 0,Y 580.304,Z 214.695,A -85,B 0,C 180,E1 -1982.772,E2 -1982.772} C_VEL
LIN {X 0,Y 580.313,Z 214.701,A -85,B 0,C 180,E1 -1985.555,E2 -1985.555} C_VEL
LIN {X 0,Y 580.303,Z 214.694,A -85,B 0,C 180,E1 -1988.351,E2 -1988.351} C_VEL
LIN {X 0,Y 580.272,Z 214.702,A -85,B 0,C 180,E1 -1991.186,E2 -1991.186} C_VEL
LIN {X 0,Y 580.317,Z 214.696,A -85,B 0,C 180,E1 -1994.011,E2 -1994.011} C_VEL
LIN {X 0,Y 580.282,Z 214.697,A -85,B 0,C 180,E1 -1996.91,E2 -1996.91} C_VEL
LIN {X 0,Y 580.279,Z 214.707,A -85,B 0,C 180,E1 -1999.817,E2 -1999.817} C_VEL
LIN {X 0,Y 580.259,Z 214.703,A -85,B 0,C 180,E1 -2001.302,E2 -2001.302} C_VEL
LIN {X 0,Y 579.574,Z 214.795,A -85,B 0,C 180,E1 -2001.881,E2 -2001.881} C_VEL
LIN {X 0,Y 576.715,Z 215.146,A -85,B 0,C 180,E1 -2002.822,E2 -2002.822} C_VEL
LIN {X 0,Y 574.32,Z 215.447,A -85,B 0,C 180,E1 -2003.579,E2 -2003.579} C_VEL
LIN {X 0,Y 573.304,Z 215.574,A -85,B 0,C 180,E1 -2004.164,E2 -2004.164} C_VEL
LIN {X 0,Y 573.227,Z 215.581,A -85,B 0,C 180,E1 -2004.361,E2 -2004.361} C_VEL
LIN {X 0,Y 573.254,Z 215.71,A -85,B 0,C 180,E1 -2005.403,E2 -2005.403} C_VEL
LIN {X 0,Y 573.644,Z 220.289,A -85,B 0,C 180,E1 -2006.164,E2 -2006.164} C_VEL
LIN {X 0,Y 573.45,Z 238.229,A -85,B 0,C 180,E1 -2009.147,E2 -2009.147} C_VEL
LIN {X 0,Y 573.284,Z 254.316,A -85,B 0,C 180,E1 -2011.805,E2 -2011.805} C_VEL
LIN {X 0,Y 573.354,Z 256.977,A -85,B 0,C 180,E1 -2012.202,E2 -2012.202} C_VEL
LIN {X 0,Y 574.041,Z 262.698,A -85,B 0,C 180,E1 -2012.316,E2 -2012.316} C_VEL
LIN {X 0,Y 573.895,Z 363.609,A -85,B 0,C 180,E1 -2013.601,E2 -2013.601} C_VEL
LIN {X 0,Y 573.783,Z 376.428,A -85,B 0,C 180,E1 -2013.89,E2 -2013.89} C_VEL
LIN {X 0,Y 573.707,Z 389.195,A -85,B 0,C 180,E1 -2014.336,E2 -2014.336} C_VEL
LIN {X 0,Y 573.584,Z 401.096,A -85,B 0,C 180,E1 -2014.889,E2 -2014.889} C_VEL
LIN {X 0,Y 573.44,Z 412.625,A -85,B 0,C 180,E1 -2015.594,E2 -2015.594} C_VEL
LIN {X 0,Y 573.358,Z 422.75,A -85,B 0,C 180,E1 -2016.359,E2 -2016.359} C_VEL
LIN {X 0,Y 573.244,Z 432.549,A -85,B 0,C 180,E1 -2017.282,E2 -2017.282} C_VEL
LIN {X 0,Y 573.149,Z 440.386,A -85,B 0,C 180,E1 -2018.174,E2 -2018.174} C_VEL
LIN {X 0,Y 573.093,Z 447.999,A -85,B 0,C 180,E1 -2019.236,E2 -2019.236} C_VEL
LIN {X 0,Y 573.032,Z 453.971,A -85,B 0,C 180,E1 -2020.279,E2 -2020.279} C_VEL
LIN {X 0,Y 573.025,Z 459.341,A -85,B 0,C 180,E1 -2021.465,E2 -2021.465} C_VEL
LIN {X 0,Y 572.975,Z 463.22,A -85,B 0,C 180,E1 -2022.615,E2 -2022.615} C_VEL
LIN {X 0,Y 572.925,Z 465.644,A -85,B 0,C 180,E1 -2023.638,E2 -2023.638} C_VEL
LIN {X 0,Y 572.939,Z 467.175,A -85,B 0,C 180,E1 -2024.649,E2 -2024.649} C_VEL
LIN {X 0,Y 572.938,Z 467.898,A -85,B 0,C 180,E1 -2025.64,E2 -2025.64} C_VEL
LIN {X 0,Y 572.923,Z 467.838,A -85,B 0,C 180,E1 -2026.614,E2 -2026.614} C_VEL
LIN {X 0,Y 572.972,Z 467.024,A -85,B 0,C 180,E1 -2027.577,E2 -2027.577} C_VEL
LIN {X 0,Y 572.965,Z 465.512,A -85,B 0,C 180,E1 -2028.522,E2 -2028.522} C_VEL
LIN {X 0,Y 572.984,Z 463.167,A -85,B 0,C 180,E1 -2029.494,E2 -2029.494} C_VEL
LIN {X 0,Y 573.004,Z 459.501,A -85,B 0,C 180,E1 -2030.585,E2 -2030.585} C_VEL
LIN {X 0,Y 573.041,Z 454.526,A -85,B 0,C 180,E1 -2031.701,E2 -2031.701} C_VEL
LIN {X 0,Y 573.077,Z 448.062,A -85,B 0,C 180,E1 -2032.844,E2 -2032.844} C_VEL
LIN {X 0,Y 573.155,Z 440.137,A -85,B 0,C 180,E1 -2033.946,E2 -2033.946} C_VEL
LIN {X 0,Y 573.221,Z 432.485,A -85,B 0,C 180,E1 -2034.815,E2 -2034.815} C_VEL
LIN {X 0,Y 573.352,Z 422.144,A -85,B 0,C 180,E1 -2035.782,E2 -2035.782} C_VEL
LIN {X 0,Y 573.455,Z 412.104,A -85,B 0,C 180,E1 -2036.532,E2 -2036.532} C_VEL
LIN {X 0,Y 573.594,Z 400.678,A -85,B 0,C 180,E1 -2037.222,E2 -2037.222} C_VEL
LIN {X 0,Y 573.696,Z 389.061,A -85,B 0,C 180,E1 -2037.76,E2 -2037.76} C_VEL
LIN {X 0,Y 573.796,Z 376.438,A -85,B 0,C 180,E1 -2038.2,E2 -2038.2} C_VEL
LIN {X 0,Y 573.894,Z 363.888,A -85,B 0,C 180,E1 -2038.485,E2 -2038.485} C_VEL
LIN {X 0,Y 573.831,Z 260.365,A -85,B 0,C 180,E1 -2039.809,E2 -2039.809} C_VEL
LIN {X 0,Y 573.326,Z 257.199,A -85,B 0,C 180,E1 -2039.876,E2 -2039.876} C_VEL
LIN {X 0,Y 573.298,Z 255.976,A -85,B 0,C 180,E1 -2040.012,E2 -2040.012} C_VEL
LIN {X 0,Y 573.461,Z 238.85,A -85,B 0,C 180,E1 -2042.839,E2 -2042.839} C_VEL
LIN {X 0,Y 573.634,Z 221.384,A -85,B 0,C 180,E1 -2045.77,E2 -2045.77} C_VEL
LIN {X 0,Y 573.501,Z 216.954,A -85,B 0,C 180,E1 -2046.532,E2 -2046.532} C_VEL
LIN {X 0,Y 573.262,Z 215.63,A -85,B 0,C 180,E1 -2046.828,E2 -2046.828} C_VEL
LIN {X 0,Y 573.188,Z 215.586,A -85,B 0,C 180,E1 -2049.923,E2 -2049.923} C_VEL
LIN {X 0,Y 573.186,Z 215.582,A -85,B 0,C 180,E1 -2052.986,E2 -2052.986} C_VEL
LIN {X 0,Y 573.214,Z 215.577,A -85,B 0,C 180,E1 -2055.807,E2 -2055.807} C_VEL
LIN {X 0,Y 573.253,Z 215.581,A -85,B 0,C 180,E1 -2058.707,E2 -2058.707} C_VEL
LIN {X 0,Y 573.235,Z 215.574,A -85,B 0,C 180,E1 -2061.541,E2 -2061.541} C_VEL
LIN {X 0,Y 573.248,Z 215.575,A -85,B 0,C 180,E1 -2064.373,E2 -2064.373} C_VEL
LIN {X 0,Y 573.248,Z 215.578,A -85,B 0,C 180,E1 -2067.19,E2 -2067.19} C_VEL
LIN {X 0,Y 573.236,Z 215.573,A -85,B 0,C 180,E1 -2070.001,E2 -2070.001} C_VEL
LIN {X 0,Y 573.247,Z 215.578,A -85,B 0,C 180,E1 -2072.812,E2 -2072.812} C_VEL
LIN {X 0,Y 573.248,Z 215.576,A -85,B 0,C 180,E1 -2075.63,E2 -2075.63} C_VEL
LIN {X 0,Y 573.236,Z 215.574,A -85,B 0,C 180,E1 -2078.461,E2 -2078.461} C_VEL
LIN {X 0,Y 573.248,Z 215.582,A -85,B 0,C 180,E1 -2081.314,E2 -2081.314} C_VEL
LIN {X 0,Y 573.216,Z 215.576,A -85,B 0,C 180,E1 -2084.432,E2 -2084.432} C_VEL
LIN {X 0,Y 573.187,Z 215.583,A -85,B 0,C 180,E1 -2087.115,E2 -2087.115} C_VEL
LIN {X 0,Y 573.19,Z 215.583,A -85,B 0,C 180,E1 -2090.08,E2 -2090.08} C_VEL
LIN {X 0,Y 573.173,Z 215.583,A -85,B 0,C 180,E1 -2092.341,E2 -2092.341} C_VEL
LIN {X 0,Y 573.213,Z 215.576,A -85,B 0,C 180,E1 -2094.886,E2 -2094.886} C_VEL
LIN {X 0,Y 573.225,Z 215.582,A -85,B 0,C 180,E1 -2097.769,E2 -2097.769} C_VEL
LIN {X 0,Y 573.211,Z 215.585,A -85,B 0,C 180,E1 -2100.179,E2 -2100.179} C_VEL
LIN {X 0,Y 573.203,Z 215.58,A -85,B 0,C 180,E1 -2102.649,E2 -2102.649} C_VEL
LIN {X 0,Y 573.212,Z 215.576,A -85,B 0,C 180,E1 -2105.188,E2 -2105.188} C_VEL
LIN {X 0,Y 573.185,Z 215.583,A -85,B 0,C 180,E1 -2107.812,E2 -2107.812} C_VEL
LIN {X 0,Y 573.217,Z 215.584,A -85,B 0,C 180,E1 -2110.534,E2 -2110.534} C_VEL
LIN {X 0,Y 573.199,Z 215.578,A -85,B 0,C 180,E1 -2113.364,E2 -2113.364} C_VEL
LIN {X 0,Y 573.208,Z 215.583,A -85,B 0,C 180,E1 -2116.336,E2 -2116.336} C_VEL
LIN {X 0,Y 573.233,Z 215.574,A -85,B 0,C 180,E1 -2119.483,E2 -2119.483} C_VEL
LIN {X 0,Y 573.199,Z 215.58,A -85,B 0,C 180,E1 -2122.199,E2 -2122.199} C_VEL
LIN {X 0,Y 573.232,Z 215.584,A -85,B 0,C 180,E1 -2124.822,E2 -2124.822} C_VEL
LIN {X 0,Y 573.223,Z 215.575,A -85,B 0,C 180,E1 -2127.777,E2 -2127.777} C_VEL
LIN {X 0,Y 573.233,Z 215.577,A -85,B 0,C 180,E1 -2130.64,E2 -2130.64} C_VEL
LIN {X 0,Y 573.209,Z 215.582,A -85,B 0,C 180,E1 -2133.514,E2 -2133.514} C_VEL
LIN {X 0,Y 573.206,Z 215.577,A -85,B 0,C 180,E1 -2136.14,E2 -2136.14} C_VEL
LIN {X 0,Y 573.235,Z 215.575,A -85,B 0,C 180,E1 -2138.715,E2 -2138.715} C_VEL
LIN {X 0,Y 573.206,Z 215.588,A -85,B 0,C 180,E1 -2141.417,E2 -2141.417} C_VEL
LIN {X 0,Y 573.231,Z 215.583,A -85,B 0,C 180,E1 -2143.627,E2 -2143.627} C_VEL
LIN {X 0,Y 573.261,Z 215.577,A -85,B 0,C 180,E1 -2145.813,E2 -2145.813} C_VEL
LIN {X 0,Y 573.258,Z 215.571,A -85,B 0,C 180,E1 -2148.751,E2 -2148.751} C_VEL
LIN {X 0,Y 573.274,Z 215.575,A -85,B 0,C 180,E1 -2151.546,E2 -2151.546} C_VEL
LIN {X 0,Y 573.281,Z 215.571,A -85,B 0,C 180,E1 -2154.377,E2 -2154.377} C_VEL
LIN {X 0,Y 573.309,Z 215.574,A -85,B 0,C 180,E1 -2157.897,E2 -2157.897} C_VEL
LIN {X 0,Y 573.328,Z 215.563,A -85,B 0,C 180,E1 -2160.707,E2 -2160.707} C_VEL
LIN {X 0,Y 573.297,Z 215.567,A -85,B 0,C 180,E1 -2162.815,E2 -2162.815} C_VEL
LIN {X 0,Y 573.269,Z 215.571,A -85,B 0,C 180,E1 -2165.633,E2 -2165.633} C_VEL
LIN {X 0,Y 573.246,Z 215.581,A -85,B 0,C 180,E1 -2168.464,E2 -2168.464} C_VEL
LIN {X 0,Y 573.284,Z 215.568,A -85,B 0,C 180,E1 -2171.316,E2 -2171.316} C_VEL
LIN {X 0,Y 573.268,Z 215.578,A -85,B 0,C 180,E1 -2174.417,E2 -2174.417} C_VEL
LIN {X 0,Y 573.26,Z 215.574,A -85,B 0,C 180,E1 -2177.115,E2 -2177.115} C_VEL
LIN {X 0,Y 573.245,Z 215.574,A -85,B 0,C 180,E1 -2180.08,E2 -2180.08} C_VEL
LIN {X 0,Y 573.232,Z 215.577,A -85,B 0,C 180,E1 -2182.341,E2 -2182.341} C_VEL
LIN {X 0,Y 573.239,Z 215.576,A -85,B 0,C 180,E1 -2185.414,E2 -2185.414} C_VEL
LIN {X 0,Y 573.214,Z 215.576,A -85,B 0,C 180,E1 -2188.021,E2 -2188.021} C_VEL
LIN {X 0,Y 573.243,Z 215.573,A -85,B 0,C 180,E1 -2190.179,E2 -2190.179} C_VEL
LIN {X 0,Y 573.26,Z 215.573,A -85,B 0,C 180,E1 -2192.648,E2 -2192.648} C_VEL
LIN {X 0,Y 573.204,Z 215.587,A -85,B 0,C 180,E1 -2195.191,E2 -2195.191} C_VEL
LIN {X 0,Y 573.243,Z 215.576,A -85,B 0,C 180,E1 -2197.81,E2 -2197.81} C_VEL
LIN {X 0,Y 573.263,Z 215.57,A -85,B 0,C 180,E1 -2200.526,E2 -2200.526} C_VEL
LIN {X 0,Y 573.22,Z 215.584,A -85,B 0,C 180,E1 -2203.665,E2 -2203.665} C_VEL
LIN {X 0,Y 573.215,Z 215.576,A -85,B 0,C 180,E1 -2206.638,E2 -2206.638} C_VEL
LIN {X 0,Y 573.261,Z 215.576,A -85,B 0,C 180,E1 -2209.475,E2 -2209.475} C_VEL
LIN {X 0,Y 573.242,Z 215.577,A -85,B 0,C 180,E1 -2212.192,E2 -2212.192} C_VEL
LIN {X 0,Y 573.234,Z 215.575,A -85,B 0,C 180,E1 -2215.231,E2 -2215.231} C_VEL
LIN {X 0,Y 573.259,Z 215.577,A -85,B 0,C 180,E1 -2217.773,E2 -2217.773} C_VEL
LIN {X 0,Y 573.252,Z 215.575,A -85,B 0,C 180,E1 -2220.633,E2 -2220.633} C_VEL
LIN {X 0,Y 573.223,Z 215.577,A -85,B 0,C 180,E1 -2223.022,E2 -2223.022} C_VEL
LIN {X 0,Y 573.229,Z 215.577,A -85,B 0,C 180,E1 -2225.363,E2 -2225.363} C_VEL
LIN {X 0,Y 573.282,Z 215.754,A -85,B 0,C 180,E1 -2227.663,E2 -2227.663} C_VEL
LIN {X 0,Y 573.895,Z 220.488,A -85,B 0,C 180,E1 -2228.445,E2 -2228.445} C_VEL
LIN {X 0,Y 573.668,Z 239.844,A -85,B 0,C 180,E1 -2231.425,E2 -2231.425} C_VEL
LIN {X 0,Y 573.432,Z 259.15,A -85,B 0,C 180,E1 -2234.357,E2 -2234.357} C_VEL
LIN {X 0,Y 573.371,Z 271.279,A -85,B 0,C 180,E1 -2236.148,E2 -2236.148} C_VEL
